LIN {X 0,Y 122.05,Z 340.248,A -85,B 0,C 180,E1 -25543.266,E2 -25543.266} C_VEL
LIN {X 0,Y 122.28,Z 340.237,A -85,B 0,C 180,E1 -25547.692,E2 -25547.692} C_VEL
LIN {X 0,Y 122.383,Z 340.24,A -85,B 0,C 180,E1 -25550.079,E2 -25550.079} C_VEL
LIN {X 0,Y 122.55,Z 340.186,A -85,B 0,C 180,E1 -25556.712,E2 -25556.712} C_VEL
LIN {X 0,Y 123.014,Z 340.16,A -85,B 0,C 180,E1 -25559.999,E2 -25559.999} C_VEL
LIN {X 0,Y 122.403,Z 340.204,A -85,B 0,C 180,E1 -25566.593,E2 -25566.593} C_VEL
LIN {X 0,Y 122.39,Z 340.237,A -85,B 0,C 180,E1 -25569.919,E2 -25569.919} C_VEL
LIN {X 0,Y 122.183,Z 340.246,A -85,B 0,C 180,E1 -25573.301,E2 -25573.301} C_VEL
LIN {X 0,Y 122.015,Z 340.287,A -85,B 0,C 180,E1 -25580.218,E2 -25580.218} C_VEL
LIN {X 0,Y 121.969,Z 340.291,A -85,B 0,C 180,E1 -25586.063,E2 -25586.063} C_VEL
LIN {X 0,Y 121.96,Z 340.291,A -85,B 0,C 180,E1 -25586.41,E2 -25586.41} C_VEL
LIN {X 0,Y 122.812,Z 342.955,A -85,B 0,C 180,E1 -25587.394,E2 -25587.394} C_VEL
LIN {X 0,Y 124.787,Z 345.128,A -85,B 0,C 180,E1 -25588.996,E2 -25588.996} C_VEL
LIN {X 0,Y 125.918,Z 346.004,A -85,B 0,C 180,E1 -25589.828,E2 -25589.828} C_VEL
LIN {X 0,Y 127.875,Z 349.273,A -85,B 0,C 180,E1 -25591.359,E2 -25591.359} C_VEL
LIN {X 0,Y 129.557,Z 351.048,A -85,B 0,C 180,E1 -25592.505,E2 -25592.505} C_VEL
LIN {X 0,Y 132.081,Z 354.649,A -85,B 0,C 180,E1 -25594.201,E2 -25594.201} C_VEL
LIN {X 0,Y 137.883,Z 363.38,A -85,B 0,C 180,E1 -25597.708,E2 -25597.708} C_VEL
LIN {X 0,Y 140.737,Z 368.366,A -85,B 0,C 180,E1 -25599.3,E2 -25599.3} C_VEL
LIN {X 0,Y 145.029,Z 378.064,A -85,B 0,C 180,E1 -25601.652,E2 -25601.652} C_VEL
LIN {X 0,Y 149.532,Z 390.716,A -85,B 0,C 180,E1 -25604.048,E2 -25604.048} C_VEL
LIN {X 0,Y 150.03,Z 393.35,A -85,B 0,C 180,E1 -25604.376,E2 -25604.376} C_VEL
LIN {X 0,Y 150.303,Z 399.971,A -85,B 0,C 180,E1 -25604.873,E2 -25604.873} C_VEL
LIN {X 0,Y 147.38,Z 443.847,A -85,B 0,C 180,E1 -25606.752,E2 -25606.752} C_VEL
LIN {X 0,Y 145.548,Z 457.609,A -85,B 0,C 180,E1 -25607.822,E2 -25607.822} C_VEL
LIN {X 0,Y 142.923,Z 470.589,A -85,B 0,C 180,E1 -25609.345,E2 -25609.345} C_VEL
LIN {X 0,Y 140.074,Z 481.613,A -85,B 0,C 180,E1 -25611.162,E2 -25611.162} C_VEL
LIN {X 0,Y 136.463,Z 493.143,A -85,B 0,C 180,E1 -25613.685,E2 -25613.685} C_VEL
LIN {X 0,Y 132.834,Z 503.54,A -85,B 0,C 180,E1 -25616.71,E2 -25616.71} C_VEL
LIN {X 0,Y 129.048,Z 513.69,A -85,B 0,C 180,E1 -25620.653,E2 -25620.653} C_VEL
LIN {X 0,Y 126.136,Z 521.23,A -85,B 0,C 180,E1 -25624.42,E2 -25624.42} C_VEL
LIN {X 0,Y 123.255,Z 528.616,A -85,B 0,C 180,E1 -25629.125,E2 -25629.125} C_VEL
LIN {X 0,Y 121.393,Z 533.602,A -85,B 0,C 180,E1 -25633.176,E2 -25633.176} C_VEL
LIN {X 0,Y 120.07,Z 538.442,A -85,B 0,C 180,E1 -25638.181,E2 -25638.181} C_VEL
LIN {X 0,Y 119.418,Z 542.133,A -85,B 0,C 180,E1 -25643.243,E2 -25643.243} C_VEL
LIN {X 0,Y 119.284,Z 544.029,A -85,B 0,C 180,E1 -25646.625,E2 -25646.625} C_VEL
LIN {X 0,Y 119.416,Z 545.463,A -85,B 0,C 180,E1 -25650.002,E2 -25650.002} C_VEL
LIN {X 0,Y 119.285,Z 546.45,A -85,B 0,C 180,E1 -25653.38,E2 -25653.38} C_VEL
LIN {X 0,Y 119.418,Z 547.051,A -85,B 0,C 180,E1 -25656.762,E2 -25656.762} C_VEL
LIN {X 0,Y 119.841,Z 547.27,A -85,B 0,C 180,E1 -25660.135,E2 -25660.135} C_VEL
LIN {X 0,Y 120.581,Z 547.087,A -85,B 0,C 180,E1 -25663.484,E2 -25663.484} C_VEL
LIN {X 0,Y 123.214,Z 545.523,A -85,B 0,C 180,E1 -25670.015,E2 -25670.015} C_VEL
LIN {X 0,Y 125.186,Z 544.168,A -85,B 0,C 180,E1 -25673.143,E2 -25673.143} C_VEL
LIN {X 0,Y 128.786,Z 541.327,A -85,B 0,C 180,E1 -25677.638,E2 -25677.638} C_VEL
LIN {X 0,Y 133.187,Z 537.486,A -85,B 0,C 180,E1 -25681.851,E2 -25681.851} C_VEL
LIN {X 0,Y 138.133,Z 532.546,A -85,B 0,C 180,E1 -25685.813,E2 -25685.813} C_VEL
LIN {X 0,Y 142.88,Z 527.3,A -85,B 0,C 180,E1 -25688.983,E2 -25688.983} C_VEL
LIN {X 0,Y 145.171,Z 524.1,A -85,B 0,C 180,E1 -25690.738,E2 -25690.738} C_VEL
LIN {X 0,Y 147.635,Z 518.574,A -85,B 0,C 180,E1 -25693.817,E2 -25693.817} C_VEL
LIN {X 0,Y 150.241,Z 512.543,A -85,B 0,C 180,E1 -25696.658,E2 -25696.658} C_VEL
LIN {X 0,Y 152.654,Z 508.469,A -85,B 0,C 180,E1 -25698.003,E2 -25698.003} C_VEL
LIN {X 0,Y 158.799,Z 498.626,A -85,B 0,C 180,E1 -25700.264,E2 -25700.264} C_VEL
LIN {X 0,Y 163.979,Z 488.786,A -85,B 0,C 180,E1 -25701.958,E2 -25701.958} C_VEL
LIN {X 0,Y 168.663,Z 478.109,A -85,B 0,C 180,E1 -25703.336,E2 -25703.336} C_VEL
LIN {X 0,Y 172.737,Z 466.399,A -85,B 0,C 180,E1 -25704.463,E2 -25704.463} C_VEL
LIN {X 0,Y 176.127,Z 453.278,A -85,B 0,C 180,E1 -25705.359,E2 -25705.359} C_VEL
LIN {X 0,Y 178.296,Z 439.911,A -85,B 0,C 180,E1 -25705.945,E2 -25705.945} C_VEL
LIN {X 0,Y 179.546,Z 425.717,A -85,B 0,C 180,E1 -25706.435,E2 -25706.435} C_VEL
LIN {X 0,Y 176.176,Z 416.595,A -85,B 0,C 180,E1 -25709.345,E2 -25709.345} C_VEL
LIN {X 0,Y 172.659,Z 408.352,A -85,B 0,C 180,E1 -25712.763,E2 -25712.763} C_VEL
LIN {X 0,Y 170.883,Z 404.467,A -85,B 0,C 180,E1 -25714.722,E2 -25714.722} C_VEL
LIN {X 0,Y 168.198,Z 398.886,A -85,B 0,C 180,E1 -25718.144,E2 -25718.144} C_VEL
LIN {X 0,Y 165.774,Z 394.965,A -85,B 0,C 180,E1 -25721.94,E2 -25721.94} C_VEL
LIN {X 0,Y 163.21,Z 390.77,A -85,B 0,C 180,E1 -25728.198,E2 -25728.198} C_VEL
LIN {X 0,Y 162.94,Z 389.949,A -85,B 0,C 180,E1 -25729.438,E2 -25729.438} C_VEL
LIN {X 0,Y 162.487,Z 389.493,A -85,B 0,C 180,E1 -25737.521,E2 -25737.521} C_VEL
LIN {X 0,Y 163.191,Z 389.938,A -85,B 0,C 180,E1 -25740.849,E2 -25740.849} C_VEL
LIN {X 0,Y 164.624,Z 393.257,A -85,B 0,C 180,E1 -25745.205,E2 -25745.205} C_VEL
LIN {X 0,Y 165.872,Z 394.947,A -85,B 0,C 180,E1 -25747.626,E2 -25747.626} C_VEL
LIN {X 0,Y 168.581,Z 399.566,A -85,B 0,C 180,E1 -25751.803,E2 -25751.803} C_VEL
LIN {X 0,Y 171.09,Z 403.702,A -85,B 0,C 180,E1 -25754.801,E2 -25754.801} C_VEL
LIN {X 0,Y 174.389,Z 409.476,A -85,B 0,C 180,E1 -25758.124,E2 -25758.124} C_VEL
LIN {X 0,Y 178.433,Z 417.155,A -85,B 0,C 180,E1 -25761.594,E2 -25761.594} C_VEL
LIN {X 0,Y 179.997,Z 420.592,A -85,B 0,C 180,E1 -25762.831,E2 -25762.831} C_VEL
LIN {X 0,Y 177.989,Z 440.073,A -85,B 0,C 180,E1 -25763.488,E2 -25763.488} C_VEL
LIN {X 0,Y 175.562,Z 452.452,A -85,B 0,C 180,E1 -25764.12,E2 -25764.12} C_VEL
LIN {X 0,Y 172.425,Z 464.153,A -85,B 0,C 180,E1 -25765.081,E2 -25765.081} C_VEL
LIN {X 0,Y 168.495,Z 475.082,A -85,B 0,C 180,E1 -25766.26,E2 -25766.26} C_VEL
LIN {X 0,Y 163.484,Z 486.45,A -85,B 0,C 180,E1 -25767.972,E2 -25767.972} C_VEL
LIN {X 0,Y 157.496,Z 497.496,A -85,B 0,C 180,E1 -25770.163,E2 -25770.163} C_VEL
LIN {X 0,Y 151.902,Z 506.082,A -85,B 0,C 180,E1 -25772.393,E2 -25772.393} C_VEL
LIN {X 0,Y 144.957,Z 515.194,A -85,B 0,C 180,E1 -25775.578,E2 -25775.578} C_VEL
LIN {X 0,Y 138.28,Z 522.741,A -85,B 0,C 180,E1 -25779.186,E2 -25779.186} C_VEL
LIN {X 0,Y 133.244,Z 527.718,A -85,B 0,C 180,E1 -25782.399,E2 -25782.399} C_VEL
LIN {X 0,Y 127.839,Z 532.518,A -85,B 0,C 180,E1 -25786.589,E2 -25786.589} C_VEL
LIN {X 0,Y 123.132,Z 536.152,A -85,B 0,C 180,E1 -25791.106,E2 -25791.106} C_VEL
LIN {X 0,Y 119.732,Z 538.422,A -85,B 0,C 180,E1 -25795.264,E2 -25795.264} C_VEL
LIN {X 0,Y 116.136,Z 540.307,A -85,B 0,C 180,E1 -25801.042,E2 -25801.042} C_VEL
LIN {X 0,Y 114.553,Z 540.859,A -85,B 0,C 180,E1 -25804.564,E2 -25804.564} C_VEL
LIN {X 0,Y 113.341,Z 540.951,A -85,B 0,C 180,E1 -25808.455,E2 -25808.455} C_VEL
LIN {X 0,Y 112.023,Z 539.967,A -85,B 0,C 180,E1 -25815.464,E2 -25815.464} C_VEL
LIN {X 0,Y 111.847,Z 538.873,A -85,B 0,C 180,E1 -25819.132,E2 -25819.132} C_VEL
LIN {X 0,Y 112,Z 537.319,A -85,B 0,C 180,E1 -25822.788,E2 -25822.788} C_VEL
LIN {X 0,Y 112.755,Z 534.417,A -85,B 0,C 180,E1 -25827.905,E2 -25827.905} C_VEL
LIN {X 0,Y 113.998,Z 530.051,A -85,B 0,C 180,E1 -25833.532,E2 -25833.532} C_VEL
LIN {X 0,Y 116.415,Z 523.712,A -85,B 0,C 180,E1 -25839.554,E2 -25839.554} C_VEL
LIN {X 0,Y 119.322,Z 516.818,A -85,B 0,C 180,E1 -25844.494,E2 -25844.494} C_VEL
LIN {X 0,Y 122.985,Z 508.179,A -85,B 0,C 180,E1 -25849.18,E2 -25849.18} C_VEL
LIN {X 0,Y 126.582,Z 499.324,A -85,B 0,C 180,E1 -25852.868,E2 -25852.868} C_VEL
LIN {X 0,Y 130.468,Z 489.549,A -85,B 0,C 180,E1 -25855.953,E2 -25855.953} C_VEL
LIN {X 0,Y 133.97,Z 478.877,A -85,B 0,C 180,E1 -25858.597,E2 -25858.597} C_VEL
LIN {X 0,Y 137.159,Z 466.941,A -85,B 0,C 180,E1 -25860.821,E2 -25860.821} C_VEL
LIN {X 0,Y 139.723,Z 454.541,A -85,B 0,C 180,E1 -25862.516,E2 -25862.516} C_VEL
LIN {X 0,Y 141.651,Z 441.546,A -85,B 0,C 180,E1 -25863.725,E2 -25863.725} C_VEL
LIN {X 0,Y 143.075,Z 424.971,A -85,B 0,C 180,E1 -25864.573,E2 -25864.573} C_VEL
LIN {X 0,Y 145.402,Z 390.427,A -85,B 0,C 180,E1 -25866.022,E2 -25866.022} C_VEL
LIN {X 0,Y 139.668,Z 378.184,A -85,B 0,C 180,E1 -25869.068,E2 -25869.068} C_VEL
LIN {X 0,Y 133.72,Z 367.749,A -85,B 0,C 180,E1 -25872.527,E2 -25872.527} C_VEL
LIN {X 0,Y 128.591,Z 360.025,A -85,B 0,C 180,E1 -25875.873,E2 -25875.873} C_VEL
LIN {X 0,Y 125.657,Z 355.95,A -85,B 0,C 180,E1 -25878,E2 -25878} C_VEL
LIN {X 0,Y 123.056,Z 352.211,A -85,B 0,C 180,E1 -25880.085,E2 -25880.085} C_VEL
LIN {X 0,Y 120.071,Z 348.913,A -85,B 0,C 180,E1 -25882.639,E2 -25882.639} C_VEL
LIN {X 0,Y 118.959,Z 346.749,A -85,B 0,C 180,E1 -25883.786,E2 -25883.786} C_VEL
LIN {X 0,Y 116.196,Z 344.608,A -85,B 0,C 180,E1 -25886.5,E2 -25886.5} C_VEL
LIN {X 0,Y 115.012,Z 342.226,A -85,B 0,C 180,E1 -25887.985,E2 -25887.985} C_VEL
LIN {X 0,Y 114.821,Z 341.175,A -85,B 0,C 180,E1 -25888.427,E2 -25888.427} C_VEL
LIN {X 0,Y 114.802,Z 341.148,A -85,B 0,C 180,E1 -25894.625,E2 -25894.625} C_VEL
LIN {X 0,Y 114.926,Z 341.167,A -85,B 0,C 180,E1 -25898.474,E2 -25898.474} C_VEL
LIN {X 0,Y 115.072,Z 341.116,A -85,B 0,C 180,E1 -25905.859,E2 -25905.859} C_VEL
LIN {X 0,Y 115.298,Z 341.121,A -85,B 0,C 180,E1 -25909.463,E2 -25909.463} C_VEL
LIN {X 0,Y 115.476,Z 341.065,A -85,B 0,C 180,E1 -25916.51,E2 -25916.51} C_VEL
LIN {X 0,Y 115.965,Z 341.038,A -85,B 0,C 180,E1 -25919.999,E2 -25919.999} C_VEL
LIN {X 0,Y 115.346,Z 341.084,A -85,B 0,C 180,E1 -25926.999,E2 -25926.999} C_VEL
LIN {X 0,Y 115.199,Z 341.123,A -85,B 0,C 180,E1 -25932.562,E2 -25932.562} C_VEL
LIN {X 0,Y 114.967,Z 341.174,A -85,B 0,C 180,E1 -25940.462,E2 -25940.462} C_VEL
LIN {X 0,Y 115.662,Z 343.507,A -85,B 0,C 180,E1 -25941.48,E2 -25941.48} C_VEL
LIN {X 0,Y 117.756,Z 345.988,A -85,B 0,C 180,E1 -25943.732,E2 -25943.732} C_VEL
LIN {X 0,Y 119.204,Z 346.968,A -85,B 0,C 180,E1 -25945.071,E2 -25945.071} C_VEL
LIN {X 0,Y 121.032,Z 350.151,A -85,B 0,C 180,E1 -25946.861,E2 -25946.861} C_VEL
LIN {X 0,Y 123.197,Z 352.402,A -85,B 0,C 180,E1 -25948.655,E2 -25948.655} C_VEL
LIN {X 0,Y 125.78,Z 356.037,A -85,B 0,C 180,E1 -25950.712,E2 -25950.712} C_VEL
LIN {X 0,Y 127.064,Z 357.855,A -85,B 0,C 180,E1 -25951.669,E2 -25951.669} C_VEL
LIN {X 0,Y 130.283,Z 362.559,A -85,B 0,C 180,E1 -25953.916,E2 -25953.916} C_VEL
LIN {X 0,Y 135.752,Z 371.145,A -85,B 0,C 180,E1 -25957.335,E2 -25957.335} C_VEL
LIN {X 0,Y 140.282,Z 381.573,A -85,B 0,C 180,E1 -25960.057,E2 -25960.057} C_VEL
LIN {X 0,Y 144.459,Z 393.679,A -85,B 0,C 180,E1 -25962.485,E2 -25962.485} C_VEL
LIN {X 0,Y 144.944,Z 399.765,A -85,B 0,C 180,E1 -25963.06,E2 -25963.06} C_VEL
LIN {X 0,Y 141.919,Z 443.257,A -85,B 0,C 180,E1 -25964.95,E2 -25964.95} C_VEL
LIN {X 0,Y 140.094,Z 456.812,A -85,B 0,C 180,E1 -25966.017,E2 -25966.017} C_VEL
LIN {X 0,Y 137.56,Z 468.886,A -85,B 0,C 180,E1 -25967.398,E2 -25967.398} C_VEL
LIN {X 0,Y 134.572,Z 480.296,A -85,B 0,C 180,E1 -25969.25,E2 -25969.25} C_VEL
LIN {X 0,Y 131.257,Z 490.735,A -85,B 0,C 180,E1 -25971.508,E2 -25971.508} C_VEL
LIN {X 0,Y 127.278,Z 501.504,A -85,B 0,C 180,E1 -25974.568,E2 -25974.568} C_VEL
LIN {X 0,Y 123.543,Z 511.223,A -85,B 0,C 180,E1 -25978.254,E2 -25978.254} C_VEL
LIN {X 0,Y 120.389,Z 519.177,A -85,B 0,C 180,E1 -25982.162,E2 -25982.162} C_VEL
LIN {X 0,Y 117.068,Z 526.893,A -85,B 0,C 180,E1 -25987.035,E2 -25987.035} C_VEL
LIN {X 0,Y 114.566,Z 533.083,A -85,B 0,C 180,E1 -25992.141,E2 -25992.141} C_VEL
LIN {X 0,Y 113.112,Z 537.994,A -85,B 0,C 180,E1 -25997.443,E2 -25997.443} C_VEL
LIN {X 0,Y 112.342,Z 541.747,A -85,B 0,C 180,E1 -26002.815,E2 -26002.815} C_VEL
LIN {X 0,Y 112.202,Z 543.674,A -85,B 0,C 180,E1 -26006.411,E2 -26006.411} C_VEL
LIN {X 0,Y 112.331,Z 545.165,A -85,B 0,C 180,E1 -26010.003,E2 -26010.003} C_VEL
LIN {X 0,Y 112.202,Z 546.182,A -85,B 0,C 180,E1 -26013.594,E2 -26013.594} C_VEL
LIN {X 0,Y 112.826,Z 547.057,A -85,B 0,C 180,E1 -26020.773,E2 -26020.773} C_VEL
LIN {X 0,Y 113.674,Z 546.921,A -85,B 0,C 180,E1 -26024.321,E2 -26024.321} C_VEL
LIN {X 0,Y 116.54,Z 545.422,A -85,B 0,C 180,E1 -26031.215,E2 -26031.215} C_VEL
LIN {X 0,Y 121.173,Z 542.372,A -85,B 0,C 180,E1 -26037.648,E2 -26037.648} C_VEL
LIN {X 0,Y 125.585,Z 538.931,A -85,B 0,C 180,E1 -26042.119,E2 -26042.119} C_VEL
LIN {X 0,Y 130.605,Z 534.436,A -85,B 0,C 180,E1 -26046.296,E2 -26046.296} C_VEL
LIN {X 0,Y 137.277,Z 527.664,A -85,B 0,C 180,E1 -26050.751,E2 -26050.751} C_VEL
LIN {X 0,Y 143.758,Z 520.325,A -85,B 0,C 180,E1 -26054.161,E2 -26054.161} C_VEL
LIN {X 0,Y 150.791,Z 511.238,A -85,B 0,C 180,E1 -26057.231,E2 -26057.231} C_VEL
LIN {X 0,Y 152.654,Z 508.469,A -85,B 0,C 180,E1 -26058.003,E2 -26058.003} C_VEL
LIN {X 0,Y 155.049,Z 504.252,A -85,B 0,C 180,E1 -26059.256,E2 -26059.256} C_VEL
LIN {X 0,Y 157.663,Z 497.141,A -85,B 0,C 180,E1 -26061.592,E2 -26061.592} C_VEL
LIN {X 0,Y 160.083,Z 489.616,A -85,B 0,C 180,E1 -26063.725,E2 -26063.725} C_VEL
LIN {X 0,Y 162.087,Z 484.679,A -85,B 0,C 180,E1 -26064.643,E2 -26064.643} C_VEL
LIN {X 0,Y 166.644,Z 473.877,A -85,B 0,C 180,E1 -26065.861,E2 -26065.861} C_VEL
LIN {X 0,Y 170.618,Z 461.527,A -85,B 0,C 180,E1 -26066.896,E2 -26066.896} C_VEL
LIN {X 0,Y 173.736,Z 448.119,A -85,B 0,C 180,E1 -26067.641,E2 -26067.641} C_VEL
LIN {X 0,Y 175.5,Z 434.788,A -85,B 0,C 180,E1 -26068.137,E2 -26068.137} C_VEL
LIN {X 0,Y 175.969,Z 428.609,A -85,B 0,C 180,E1 -26068.386,E2 -26068.386} C_VEL
LIN {X 0,Y 172.859,Z 420.02,A -85,B 0,C 180,E1 -26071.381,E2 -26071.381} C_VEL
LIN {X 0,Y 169.949,Z 412.743,A -85,B 0,C 180,E1 -26074.578,E2 -26074.578} C_VEL
LIN {X 0,Y 167.428,Z 407.201,A -85,B 0,C 180,E1 -26077.804,E2 -26077.804} C_VEL
LIN {X 0,Y 166.423,Z 405.138,A -85,B 0,C 180,E1 -26079.288,E2 -26079.288} C_VEL
LIN {X 0,Y 164.199,Z 401.326,A -85,B 0,C 180,E1 -26083.169,E2 -26083.169} C_VEL
LIN {X 0,Y 162.181,Z 397.615,A -85,B 0,C 180,E1 -26088.755,E2 -26088.755} C_VEL
LIN {X 0,Y 161.931,Z 396.919,A -85,B 0,C 180,E1 -26090.003,E2 -26090.003} C_VEL
LIN {X 0,Y 161.725,Z 396.564,A -85,B 0,C 180,E1 -26098.228,E2 -26098.228} C_VEL
LIN {X 0,Y 162.203,Z 396.945,A -85,B 0,C 180,E1 -26100.466,E2 -26100.466} C_VEL
LIN {X 0,Y 163.599,Z 400.242,A -85,B 0,C 180,E1 -26104.929,E2 -26104.929} C_VEL
LIN {X 0,Y 164.553,Z 401.63,A -85,B 0,C 180,E1 -26106.9,E2 -26106.9} C_VEL
LIN {X 0,Y 167.015,Z 406.088,A -85,B 0,C 180,E1 -26110.993,E2 -26110.993} C_VEL
LIN {X 0,Y 169.332,Z 410.145,A -85,B 0,C 180,E1 -26113.96,E2 -26113.96} C_VEL
LIN {X 0,Y 172.088,Z 415.151,A -85,B 0,C 180,E1 -26116.936,E2 -26116.936} C_VEL
LIN {X 0,Y 176.206,Z 423.49,A -85,B 0,C 180,E1 -26120.732,E2 -26120.732} C_VEL
LIN {X 0,Y 176.439,Z 424.028,A -85,B 0,C 180,E1 -26120.932,E2 -26120.932} C_VEL
LIN {X 0,Y 174.441,Z 441.483,A -85,B 0,C 180,E1 -26121.51,E2 -26121.51} C_VEL
LIN {X 0,Y 171.775,Z 454.185,A -85,B 0,C 180,E1 -26122.182,E2 -26122.182} C_VEL
LIN {X 0,Y 167.865,Z 467.297,A -85,B 0,C 180,E1 -26123.295,E2 -26123.295} C_VEL
LIN {X 0,Y 163.346,Z 478.817,A -85,B 0,C 180,E1 -26124.642,E2 -26124.642} C_VEL
LIN {X 0,Y 158.004,Z 489.815,A -85,B 0,C 180,E1 -26126.411,E2 -26126.411} C_VEL
LIN {X 0,Y 151.981,Z 499.889,A -85,B 0,C 180,E1 -26128.522,E2 -26128.522} C_VEL
LIN {X 0,Y 145.617,Z 508.928,A -85,B 0,C 180,E1 -26131.051,E2 -26131.051} C_VEL
LIN {X 0,Y 138.684,Z 517.33,A -85,B 0,C 180,E1 -26134.212,E2 -26134.212} C_VEL
LIN {X 0,Y 131.583,Z 524.614,A -85,B 0,C 180,E1 -26138.015,E2 -26138.015} C_VEL
LIN {X 0,Y 124.487,Z 530.95,A -85,B 0,C 180,E1 -26142.781,E2 -26142.781} C_VEL
LIN {X 0,Y 119.123,Z 535.036,A -85,B 0,C 180,E1 -26147.273,E2 -26147.273} C_VEL
LIN {X 0,Y 113.347,Z 538.705,A -85,B 0,C 180,E1 -26153.714,E2 -26153.714} C_VEL
LIN {X 0,Y 109.773,Z 540.425,A -85,B 0,C 180,E1 -26159.188,E2 -26159.188} C_VEL
LIN {X 0,Y 107.982,Z 541.012,A -85,B 0,C 180,E1 -26162.894,E2 -26162.894} C_VEL
LIN {X 0,Y 106.365,Z 541.14,A -85,B 0,C 180,E1 -26167.678,E2 -26167.678} C_VEL
LIN {X 0,Y 105.029,Z 540.255,A -85,B 0,C 180,E1 -26174.472,E2 -26174.472} C_VEL
LIN {X 0,Y 104.763,Z 539.201,A -85,B 0,C 180,E1 -26178.387,E2 -26178.387} C_VEL
LIN {X 0,Y 104.857,Z 537.712,A -85,B 0,C 180,E1 -26182.294,E2 -26182.294} C_VEL
LIN {X 0,Y 105.554,Z 535.228,A -85,B 0,C 180,E1 -26187.135,E2 -26187.135} C_VEL
LIN {X 0,Y 106.911,Z 530.591,A -85,B 0,C 180,E1 -26193.766,E2 -26193.766} C_VEL
LIN {X 0,Y 109.417,Z 524.337,A -85,B 0,C 180,E1 -26200.171,E2 -26200.171} C_VEL
LIN {X 0,Y 112.45,Z 517.538,A -85,B 0,C 180,E1 -26205.401,E2 -26205.401} C_VEL
LIN {X 0,Y 116.317,Z 509.064,A -85,B 0,C 180,E1 -26210.327,E2 -26210.327} C_VEL
LIN {X 0,Y 120.084,Z 500.345,A -85,B 0,C 180,E1 -26214.182,E2 -26214.182} C_VEL
LIN {X 0,Y 124.021,Z 490.76,A -85,B 0,C 180,E1 -26217.412,E2 -26217.412} C_VEL
LIN {X 0,Y 127.816,Z 480.285,A -85,B 0,C 180,E1 -26220.112,E2 -26220.112} C_VEL
LIN {X 0,Y 131.152,Z 468.802,A -85,B 0,C 180,E1 -26222.4,E2 -26222.4} C_VEL
LIN {X 0,Y 133.852,Z 456.913,A -85,B 0,C 180,E1 -26224.133,E2 -26224.133} C_VEL
LIN {X 0,Y 136.084,Z 443.206,A -85,B 0,C 180,E1 -26225.516,E2 -26225.516} C_VEL
LIN {X 0,Y 137.339,Z 430.812,A -85,B 0,C 180,E1 -26226.261,E2 -26226.261} C_VEL
LIN {X 0,Y 140.056,Z 392.687,A -85,B 0,C 180,E1 -26227.88,E2 -26227.88} C_VEL
LIN {X 0,Y 134.901,Z 381.566,A -85,B 0,C 180,E1 -26230.886,E2 -26230.886} C_VEL
LIN {X 0,Y 129.535,Z 372.061,A -85,B 0,C 180,E1 -26234.298,E2 -26234.298} C_VEL
LIN {X 0,Y 125.1,Z 365.244,A -85,B 0,C 180,E1 -26237.455,E2 -26237.455} C_VEL
LIN {X 0,Y 122.486,Z 361.454,A -85,B 0,C 180,E1 -26239.524,E2 -26239.524} C_VEL
LIN {X 0,Y 119.777,Z 357.638,A -85,B 0,C 180,E1 -26241.885,E2 -26241.885} C_VEL
LIN {X 0,Y 117.217,Z 354.408,A -85,B 0,C 180,E1 -26244.333,E2 -26244.333} C_VEL
LIN {X 0,Y 116.461,Z 353.066,A -85,B 0,C 180,E1 -26245.163,E2 -26245.163} C_VEL
LIN {X 0,Y 113.857,Z 350.628,A -85,B 0,C 180,E1 -26247.983,E2 -26247.983} C_VEL
LIN {X 0,Y 112.387,Z 347.844,A -85,B 0,C 180,E1 -26249.981,E2 -26249.981} C_VEL
LIN {X 0,Y 109.653,Z 346.082,A -85,B 0,C 180,E1 -26253.723,E2 -26253.723} C_VEL
LIN {X 0,Y 108.268,Z 343.712,A -85,B 0,C 180,E1 -26256.287,E2 -26256.287} C_VEL
LIN {X 0,Y 107.871,Z 342.033,A -85,B 0,C 180,E1 -26257.494,E2 -26257.494} C_VEL
LIN {X 0,Y 107.961,Z 341.997,A -85,B 0,C 180,E1 -26264.906,E2 -26264.906} C_VEL
LIN {X 0,Y 108.216,Z 341.998,A -85,B 0,C 180,E1 -26268.764,E2 -26268.764} C_VEL
LIN {X 0,Y 108.279,Z 341.973,A -85,B 0,C 180,E1 -26272.54,E2 -26272.54} C_VEL
LIN {X 0,Y 108.891,Z 341.919,A -85,B 0,C 180,E1 -26279.999,E2 -26279.999} C_VEL
LIN {X 0,Y 108.285,Z 341.965,A -85,B 0,C 180,E1 -26287.458,E2 -26287.458} C_VEL
LIN {X 0,Y 108.198,Z 342.025,A -85,B 0,C 180,E1 -26291.861,E2 -26291.861} C_VEL
LIN {X 0,Y 108.799,Z 344.324,A -85,B 0,C 180,E1 -26293.314,E2 -26293.314} C_VEL
LIN {X 0,Y 110.502,Z 346.638,A -85,B 0,C 180,E1 -26296.155,E2 -26296.155} C_VEL
LIN {X 0,Y 112.749,Z 348.094,A -85,B 0,C 180,E1 -26299.101,E2 -26299.101} C_VEL
LIN {X 0,Y 114.313,Z 351.012,A -85,B 0,C 180,E1 -26301.173,E2 -26301.173} C_VEL
LIN {X 0,Y 116.89,Z 353.611,A -85,B 0,C 180,E1 -26303.918,E2 -26303.918} C_VEL
LIN {X 0,Y 119.215,Z 357.045,A -85,B 0,C 180,E1 -26306.24,E2 -26306.24} C_VEL
LIN {X 0,Y 120.52,Z 358.544,A -85,B 0,C 180,E1 -26307.395,E2 -26307.395} C_VEL
LIN {X 0,Y 124.501,Z 364.347,A -85,B 0,C 180,E1 -26310.709,E2 -26310.709} C_VEL
LIN {X 0,Y 128.263,Z 370.003,A -85,B 0,C 180,E1 -26313.46,E2 -26313.46} C_VEL
LIN {X 0,Y 132.251,Z 376.864,A -85,B 0,C 180,E1 -26316.124,E2 -26316.124} C_VEL
LIN {X 0,Y 136.104,Z 386.284,A -85,B 0,C 180,E1 -26318.644,E2 -26318.644} C_VEL
LIN {X 0,Y 139.507,Z 396.653,A -85,B 0,C 180,E1 -26320.814,E2 -26320.814} C_VEL
LIN {X 0,Y 139.582,Z 402.148,A -85,B 0,C 180,E1 -26321.23,E2 -26321.23} C_VEL
LIN {X 0,Y 136.517,Z 443.449,A -85,B 0,C 180,E1 -26323.057,E2 -26323.057} C_VEL
LIN {X 0,Y 134.636,Z 456.775,A -85,B 0,C 180,E1 -26324.135,E2 -26324.135} C_VEL
LIN {X 0,Y 131.854,Z 469.366,A -85,B 0,C 180,E1 -26325.611,E2 -26325.611} C_VEL
LIN {X 0,Y 128.732,Z 480.582,A -85,B 0,C 180,E1 -26327.503,E2 -26327.503} C_VEL
LIN {X 0,Y 124.801,Z 492.239,A -85,B 0,C 180,E1 -26330.169,E2 -26330.169} C_VEL
LIN {X 0,Y 120.681,Z 502.718,A -85,B 0,C 180,E1 -26333.354,E2 -26333.354} C_VEL
LIN {X 0,Y 116.768,Z 512.141,A -85,B 0,C 180,E1 -26337.205,E2 -26337.205} C_VEL
LIN {X 0,Y 113.458,Z 519.883,A -85,B 0,C 180,E1 -26341.314,E2 -26341.314} C_VEL
LIN {X 0,Y 110.014,Z 527.43,A -85,B 0,C 180,E1 -26346.471,E2 -26346.471} C_VEL
LIN {X 0,Y 107.152,Z 534.387,A -85,B 0,C 180,E1 -26352.837,E2 -26352.837} C_VEL
LIN {X 0,Y 105.785,Z 538.963,A -85,B 0,C 180,E1 -26358.506,E2 -26358.506} C_VEL
LIN {X 0,Y 105.283,Z 541.362,A -85,B 0,C 180,E1 -26362.331,E2 -26362.331} C_VEL
LIN {X 0,Y 105.111,Z 543.32,A -85,B 0,C 180,E1 -26366.169,E2 -26366.169} C_VEL
LIN {X 0,Y 105.232,Z 544.854,A -85,B 0,C 180,E1 -26370.003,E2 -26370.003} C_VEL
LIN {X 0,Y 105.112,Z 545.913,A -85,B 0,C 180,E1 -26373.837,E2 -26373.837} C_VEL
LIN {X 0,Y 105.841,Z 546.843,A -85,B 0,C 180,E1 -26381.493,E2 -26381.493} C_VEL
LIN {X 0,Y 106.801,Z 546.74,A -85,B 0,C 180,E1 -26385.264,E2 -26385.264} C_VEL
LIN {X 0,Y 108.151,Z 546.236,A -85,B 0,C 180,E1 -26388.963,E2 -26388.963} C_VEL
LIN {X 0,Y 112.232,Z 544.023,A -85,B 0,C 180,E1 -26396.001,E2 -26396.001} C_VEL
LIN {X 0,Y 116.353,Z 541.302,A -85,B 0,C 180,E1 -26400.895,E2 -26400.895} C_VEL
LIN {X 0,Y 121.326,Z 537.588,A -85,B 0,C 180,E1 -26405.401,E2 -26405.401} C_VEL
LIN {X 0,Y 126.883,Z 532.786,A -85,B 0,C 180,E1 -26409.57,E2 -26409.57} C_VEL
LIN {X 0,Y 133.07,Z 526.753,A -85,B 0,C 180,E1 -26413.363,E2 -26413.363} C_VEL
LIN {X 0,Y 139.975,Z 519.263,A -85,B 0,C 180,E1 -26416.724,E2 -26416.724} C_VEL
LIN {X 0,Y 146.072,Z 511.636,A -85,B 0,C 180,E1 -26419.272,E2 -26419.272} C_VEL
LIN {X 0,Y 152.438,Z 502.393,A -85,B 0,C 180,E1 -26421.609,E2 -26421.609} C_VEL
LIN {X 0,Y 158.314,Z 492.142,A -85,B 0,C 180,E1 -26423.576,E2 -26423.576} C_VEL
LIN {X 0,Y 162.087,Z 484.679,A -85,B 0,C 180,E1 -26424.643,E2 -26424.643} C_VEL
LIN {X 0,Y 164.012,Z 479.628,A -85,B 0,C 180,E1 -26425.493,E2 -26425.493} C_VEL
LIN {X 0,Y 165.958,Z 471.251,A -85,B 0,C 180,E1 -26427.214,E2 -26427.214} C_VEL
LIN {X 0,Y 167.458,Z 462.549,A -85,B 0,C 180,E1 -26428.747,E2 -26428.747} C_VEL
LIN {X 0,Y 168.609,Z 456.994,A -85,B 0,C 180,E1 -26429.299,E2 -26429.299} C_VEL
LIN {X 0,Y 171.296,Z 443.775,A -85,B 0,C 180,E1 -26429.931,E2 -26429.931} C_VEL
LIN {X 0,Y 172.656,Z 431.847,A -85,B 0,C 180,E1 -26430.346,E2 -26430.346} C_VEL
LIN {X 0,Y 169.953,Z 423.974,A -85,B 0,C 180,E1 -26433.275,E2 -26433.275} C_VEL
LIN {X 0,Y 167.224,Z 416.916,A -85,B 0,C 180,E1 -26436.675,E2 -26436.675} C_VEL
LIN {X 0,Y 165.141,Z 411.961,A -85,B 0,C 180,E1 -26439.803,E2 -26439.803} C_VEL
LIN {X 0,Y 163.016,Z 408.16,A -85,B 0,C 180,E1 -26443.726,E2 -26443.726} C_VEL
LIN {X 0,Y 161.116,Z 404.213,A -85,B 0,C 180,E1 -26449.634,E2 -26449.634} C_VEL
LIN {X 0,Y 160.656,Z 403.702,A -85,B 0,C 180,E1 -26452.459,E2 -26452.459} C_VEL
LIN {X 0,Y 161.104,Z 403.741,A -85,B 0,C 180,E1 -26459.511,E2 -26459.511} C_VEL
LIN {X 0,Y 161.586,Z 405.348,A -85,B 0,C 180,E1 -26461.792,E2 -26461.792} C_VEL
LIN {X 0,Y 163.36,Z 408.499,A -85,B 0,C 180,E1 -26466.369,E2 -26466.369} C_VEL
LIN {X 0,Y 165.583,Z 412.811,A -85,B 0,C 180,E1 -26470.316,E2 -26470.316} C_VEL
LIN {X 0,Y 167.584,Z 416.516,A -85,B 0,C 180,E1 -26473.066,E2 -26473.066} C_VEL
LIN {X 0,Y 170.54,Z 422.339,A -85,B 0,C 180,E1 -26476.459,E2 -26476.459} C_VEL
LIN {X 0,Y 173.025,Z 427.558,A -85,B 0,C 180,E1 -26478.925,E2 -26478.925} C_VEL
LIN {X 0,Y 171.194,Z 442.453,A -85,B 0,C 180,E1 -26479.445,E2 -26479.445} C_VEL
LIN {X 0,Y 168.641,Z 454.043,A -85,B 0,C 180,E1 -26480.023,E2 -26480.023} C_VEL
LIN {X 0,Y 164.757,Z 466.842,A -85,B 0,C 180,E1 -26481.07,E2 -26481.07} C_VEL
LIN {X 0,Y 160.451,Z 477.689,A -85,B 0,C 180,E1 -26482.282,E2 -26482.282} C_VEL
LIN {X 0,Y 155.387,Z 488.05,A -85,B 0,C 180,E1 -26483.827,E2 -26483.827} C_VEL
LIN {X 0,Y 149.312,Z 498.308,A -85,B 0,C 180,E1 -26485.84,E2 -26485.84} C_VEL
LIN {X 0,Y 143.289,Z 506.782,A -85,B 0,C 180,E1 -26488.008,E2 -26488.008} C_VEL
LIN {X 0,Y 135.541,Z 516.03,A -85,B 0,C 180,E1 -26491.234,E2 -26491.234} C_VEL
LIN {X 0,Y 128.364,Z 523.341,A -85,B 0,C 180,E1 -26494.786,E2 -26494.786} C_VEL
LIN {X 0,Y 121.698,Z 529.175,A -85,B 0,C 180,E1 -26498.771,E2 -26498.771} C_VEL
LIN {X 0,Y 115.689,Z 533.722,A -85,B 0,C 180,E1 -26503.195,E2 -26503.195} C_VEL
LIN {X 0,Y 112.086,Z 536.104,A -85,B 0,C 180,E1 -26506.389,E2 -26506.389} C_VEL
LIN {X 0,Y 107.049,Z 538.995,A -85,B 0,C 180,E1 -26511.985,E2 -26511.985} C_VEL
LIN {X 0,Y 103.554,Z 540.544,A -85,B 0,C 180,E1 -26517.113,E2 -26517.113} C_VEL
LIN {X 0,Y 99.964,Z 541.389,A -85,B 0,C 180,E1 -26525.047,E2 -26525.047} C_VEL
LIN {X 0,Y 98.834,Z 541.172,A -85,B 0,C 180,E1 -26529.17,E2 -26529.17} C_VEL
LIN {X 0,Y 98.047,Z 540.544,A -85,B 0,C 180,E1 -26533.335,E2 -26533.335} C_VEL
LIN {X 0,Y 97.691,Z 539.523,A -85,B 0,C 180,E1 -26537.533,E2 -26537.533} C_VEL
LIN {X 0,Y 97.72,Z 538.098,A -85,B 0,C 180,E1 -26541.727,E2 -26541.727} C_VEL
LIN {X 0,Y 98.49,Z 535.37,A -85,B 0,C 180,E1 -26547.469,E2 -26547.469} C_VEL
LIN {X 0,Y 99.828,Z 531.114,A -85,B 0,C 180,E1 -26554.034,E2 -26554.034} C_VEL
LIN {X 0,Y 102.439,Z 524.96,A -85,B 0,C 180,E1 -26560.872,E2 -26560.872} C_VEL
LIN {X 0,Y 105.619,Z 518.255,A -85,B 0,C 180,E1 -26566.424,E2 -26566.424} C_VEL
LIN {X 0,Y 109.704,Z 509.929,A -85,B 0,C 180,E1 -26571.612,E2 -26571.612} C_VEL
LIN {X 0,Y 113.661,Z 501.359,A -85,B 0,C 180,E1 -26575.644,E2 -26575.644} C_VEL
LIN {X 0,Y 118.247,Z 490.765,A -85,B 0,C 180,E1 -26579.36,E2 -26579.36} C_VEL
LIN {X 0,Y 121.764,Z 481.668,A -85,B 0,C 180,E1 -26581.778,E2 -26581.778} C_VEL
LIN {X 0,Y 125.257,Z 470.492,A -85,B 0,C 180,E1 -26584.128,E2 -26584.128} C_VEL
LIN {X 0,Y 128.336,Z 457.972,A -85,B 0,C 180,E1 -26586.061,E2 -26586.061} C_VEL
LIN {X 0,Y 130.693,Z 444.534,A -85,B 0,C 180,E1 -26587.473,E2 -26587.473} C_VEL
LIN {X 0,Y 132.133,Z 431.622,A -85,B 0,C 180,E1 -26588.293,E2 -26588.293} C_VEL
LIN {X 0,Y 134.884,Z 395.035,A -85,B 0,C 180,E1 -26589.866,E2 -26589.866} C_VEL
LIN {X 0,Y 130.505,Z 385.503,A -85,B 0,C 180,E1 -26592.667,E2 -26592.667} C_VEL
LIN {X 0,Y 125.785,Z 376.91,A -85,B 0,C 180,E1 -26595.954,E2 -26595.954} C_VEL
LIN {X 0,Y 121.727,Z 370.416,A -85,B 0,C 180,E1 -26599.125,E2 -26599.125} C_VEL
LIN {X 0,Y 119.221,Z 366.73,A -85,B 0,C 180,E1 -26601.298,E2 -26601.298} C_VEL
LIN {X 0,Y 117.116,Z 363.62,A -85,B 0,C 180,E1 -26603.308,E2 -26603.308} C_VEL
LIN {X 0,Y 114.568,Z 360.07,A -85,B 0,C 180,E1 -26605.996,E2 -26605.996} C_VEL
LIN {X 0,Y 113.756,Z 359.087,A -85,B 0,C 180,E1 -26606.91,E2 -26606.91} C_VEL
LIN {X 0,Y 111.313,Z 356.145,A -85,B 0,C 180,E1 -26609.923,E2 -26609.923} C_VEL
LIN {X 0,Y 110.436,Z 354.477,A -85,B 0,C 180,E1 -26611.231,E2 -26611.231} C_VEL
LIN {X 0,Y 107.921,Z 352.543,A -85,B 0,C 180,E1 -26615.013,E2 -26615.013} C_VEL
LIN {X 0,Y 106.473,Z 349.767,A -85,B 0,C 180,E1 -26618.051,E2 -26618.051} C_VEL
LIN {X 0,Y 106.094,Z 348.921,A -85,B 0,C 180,E1 -26618.989,E2 -26618.989} C_VEL
LIN {X 0,Y 102.737,Z 346.454,A -85,B 0,C 180,E1 -26632.136,E2 -26632.136} C_VEL
LIN {X 0,Y 103.264,Z 346.379,A -85,B 0,C 180,E1 -26640.487,E2 -26640.487} C_VEL
LIN {X 0,Y 105.435,Z 348.496,A -85,B 0,C 180,E1 -26648.142,E2 -26648.142} C_VEL
LIN {X 0,Y 106.56,Z 349.064,A -85,B 0,C 180,E1 -26650.569,E2 -26650.569} C_VEL
LIN {X 0,Y 107.737,Z 351.889,A -85,B 0,C 180,E1 -26653.2,E2 -26653.2} C_VEL
LIN {X 0,Y 109.935,Z 354.097,A -85,B 0,C 180,E1 -26656.707,E2 -26656.707} C_VEL
LIN {X 0,Y 110.853,Z 354.917,A -85,B 0,C 180,E1 -26657.979,E2 -26657.979} C_VEL
LIN {X 0,Y 112.964,Z 358.201,A -85,B 0,C 180,E1 -26660.811,E2 -26660.811} C_VEL
LIN {X 0,Y 114.596,Z 359.988,A -85,B 0,C 180,E1 -26662.657,E2 -26662.657} C_VEL
LIN {X 0,Y 117.117,Z 363.548,A -85,B 0,C 180,E1 -26665.312,E2 -26665.312} C_VEL
LIN {X 0,Y 121.31,Z 369.722,A -85,B 0,C 180,E1 -26669.144,E2 -26669.144} C_VEL
LIN {X 0,Y 125.191,Z 375.902,A -85,B 0,C 180,E1 -26672.229,E2 -26672.229} C_VEL
LIN {X 0,Y 128.563,Z 382.032,A -85,B 0,C 180,E1 -26674.671,E2 -26674.671} C_VEL
LIN {X 0,Y 132.094,Z 391.319,A -85,B 0,C 180,E1 -26677.207,E2 -26677.207} C_VEL
LIN {X 0,Y 134.527,Z 399.408,A -85,B 0,C 180,E1 -26678.942,E2 -26678.942} C_VEL
LIN {X 0,Y 134.359,Z 404.188,A -85,B 0,C 180,E1 -26679.228,E2 -26679.228} C_VEL
LIN {X 0,Y 131.248,Z 443.904,A -85,B 0,C 180,E1 -26681.033,E2 -26681.033} C_VEL
LIN {X 0,Y 129.162,Z 457.475,A -85,B 0,C 180,E1 -26682.156,E2 -26682.156} C_VEL
LIN {X 0,Y 126.293,Z 469.791,A -85,B 0,C 180,E1 -26683.666,E2 -26683.666} C_VEL
LIN {X 0,Y 122.507,Z 482.461,A -85,B 0,C 180,E1 -26685.93,E2 -26685.93} C_VEL
LIN {X 0,Y 118.363,Z 493.729,A -85,B 0,C 180,E1 -26688.661,E2 -26688.661} C_VEL
LIN {X 0,Y 114.148,Z 503.855,A -85,B 0,C 180,E1 -26692.002,E2 -26692.002} C_VEL
LIN {X 0,Y 109.827,Z 513.526,A -85,B 0,C 180,E1 -26696.292,E2 -26696.292} C_VEL
LIN {X 0,Y 105.837,Z 521.939,A -85,B 0,C 180,E1 -26701.225,E2 -26701.225} C_VEL
LIN {X 0,Y 102.47,Z 529.055,A -85,B 0,C 180,E1 -26706.777,E2 -26706.777} C_VEL
LIN {X 0,Y 100.333,Z 533.88,A -85,B 0,C 180,E1 -26711.63,E2 -26711.63} C_VEL
LIN {X 0,Y 98.793,Z 538.531,A -85,B 0,C 180,E1 -26717.681,E2 -26717.681} C_VEL
LIN {X 0,Y 98.251,Z 540.977,A -85,B 0,C 180,E1 -26721.778,E2 -26721.778} C_VEL
LIN {X 0,Y 98.021,Z 542.965,A -85,B 0,C 180,E1 -26725.891,E2 -26725.891} C_VEL
LIN {X 0,Y 98.144,Z 544.531,A -85,B 0,C 180,E1 -26730.003,E2 -26730.003} C_VEL
LIN {X 0,Y 98.022,Z 545.644,A -85,B 0,C 180,E1 -26734.114,E2 -26734.114} C_VEL
LIN {X 0,Y 98.887,Z 546.63,A -85,B 0,C 180,E1 -26742.314,E2 -26742.314} C_VEL
LIN {X 0,Y 101.424,Z 546.099,A -85,B 0,C 180,E1 -26750.274,E2 -26750.274} C_VEL
LIN {X 0,Y 105.882,Z 543.955,A -85,B 0,C 180,E1 -26757.689,E2 -26757.689} C_VEL
LIN {X 0,Y 110.31,Z 541.296,A -85,B 0,C 180,E1 -26762.792,E2 -26762.792} C_VEL
LIN {X 0,Y 115.587,Z 537.647,A -85,B 0,C 180,E1 -26767.45,E2 -26767.45} C_VEL
LIN {X 0,Y 121.487,Z 532.915,A -85,B 0,C 180,E1 -26771.706,E2 -26771.706} C_VEL
LIN {X 0,Y 127.995,Z 526.958,A -85,B 0,C 180,E1 -26775.548,E2 -26775.548} C_VEL
LIN {X 0,Y 135.204,Z 519.554,A -85,B 0,C 180,E1 -26778.916,E2 -26778.916} C_VEL
LIN {X 0,Y 142.847,Z 510.361,A -85,B 0,C 180,E1 -26781.926,E2 -26781.926} C_VEL
LIN {X 0,Y 150.152,Z 499.777,A -85,B 0,C 180,E1 -26784.417,E2 -26784.417} C_VEL
LIN {X 0,Y 155.658,Z 490.298,A -85,B 0,C 180,E1 -26786.064,E2 -26786.064} C_VEL
LIN {X 0,Y 161.339,Z 478.501,A -85,B 0,C 180,E1 -26787.565,E2 -26787.565} C_VEL
LIN {X 0,Y 165.94,Z 466.164,A -85,B 0,C 180,E1 -26788.689,E2 -26788.689} C_VEL
LIN {X 0,Y 168.609,Z 456.994,A -85,B 0,C 180,E1 -26789.299,E2 -26789.299} C_VEL
LIN {X 0,Y 169.22,Z 453.238,A -85,B 0,C 180,E1 -26789.715,E2 -26789.715} C_VEL
LIN {X 0,Y 169.208,Z 447.406,A -85,B 0,C 180,E1 -26790.874,E2 -26790.874} C_VEL
LIN {X 0,Y 169.025,Z 441.512,A -85,B 0,C 180,E1 -26791.989,E2 -26791.989} C_VEL
LIN {X 0,Y 169.232,Z 437.662,A -85,B 0,C 180,E1 -26792.325,E2 -26792.325} C_VEL
LIN {X 0,Y 169.487,Z 434.94,A -85,B 0,C 180,E1 -26792.449,E2 -26792.449} C_VEL
LIN {X 0,Y 166.893,Z 427.074,A -85,B 0,C 180,E1 -26795.676,E2 -26795.676} C_VEL
LIN {X 0,Y 164.715,Z 421.114,A -85,B 0,C 180,E1 -26798.864,E2 -26798.864} C_VEL
LIN {X 0,Y 163.483,Z 418.253,A -85,B 0,C 180,E1 -26800.959,E2 -26800.959} C_VEL
LIN {X 0,Y 161.867,Z 415.009,A -85,B 0,C 180,E1 -26804.255,E2 -26804.255} C_VEL
LIN {X 0,Y 160.069,Z 410.982,A -85,B 0,C 180,E1 -26810.524,E2 -26810.524} C_VEL
LIN {X 0,Y 160.068,Z 410.711,A -85,B 0,C 180,E1 -26818.743,E2 -26818.743} C_VEL
LIN {X 0,Y 160.3,Z 411.211,A -85,B 0,C 180,E1 -26820,E2 -26820} C_VEL
LIN {X 0,Y 162.129,Z 415.272,A -85,B 0,C 180,E1 -26825.715,E2 -26825.715} C_VEL
LIN {X 0,Y 164.105,Z 419.336,A -85,B 0,C 180,E1 -26829.501,E2 -26829.501} C_VEL
LIN {X 0,Y 166.097,Z 423.32,A -85,B 0,C 180,E1 -26832.447,E2 -26832.447} C_VEL
LIN {X 0,Y 169.225,Z 429.895,A -85,B 0,C 180,E1 -26836.203,E2 -26836.203} C_VEL
LIN {X 0,Y 169.81,Z 431.277,A -85,B 0,C 180,E1 -26836.841,E2 -26836.841} C_VEL
LIN {X 0,Y 167.863,Z 444.737,A -85,B 0,C 180,E1 -26837.336,E2 -26837.336} C_VEL
LIN {X 0,Y 164.86,Z 457.215,A -85,B 0,C 180,E1 -26838.04,E2 -26838.04} C_VEL
LIN {X 0,Y 160.792,Z 469.442,A -85,B 0,C 180,E1 -26839.053,E2 -26839.053} C_VEL
LIN {X 0,Y 156.359,Z 479.791,A -85,B 0,C 180,E1 -26840.231,E2 -26840.231} C_VEL
LIN {X 0,Y 150.652,Z 490.627,A -85,B 0,C 180,E1 -26841.914,E2 -26841.914} C_VEL
LIN {X 0,Y 144.182,Z 500.644,A -85,B 0,C 180,E1 -26843.939,E2 -26843.939} C_VEL
LIN {X 0,Y 137.292,Z 509.621,A -85,B 0,C 180,E1 -26846.382,E2 -26846.382} C_VEL
LIN {X 0,Y 131.198,Z 516.41,A -85,B 0,C 180,E1 -26848.824,E2 -26848.824} C_VEL
LIN {X 0,Y 124.344,Z 523.074,A -85,B 0,C 180,E1 -26852.022,E2 -26852.022} C_VEL
LIN {X 0,Y 117.248,Z 529.018,A -85,B 0,C 180,E1 -26855.978,E2 -26855.978} C_VEL
LIN {X 0,Y 110.802,Z 533.658,A -85,B 0,C 180,E1 -26860.432,E2 -26860.432} C_VEL
LIN {X 0,Y 106.889,Z 536.083,A -85,B 0,C 180,E1 -26863.673,E2 -26863.673} C_VEL
LIN {X 0,Y 100.887,Z 539.276,A -85,B 0,C 180,E1 -26870.023,E2 -26870.023} C_VEL
LIN {X 0,Y 97.476,Z 540.664,A -85,B 0,C 180,E1 -26874.771,E2 -26874.771} C_VEL
LIN {X 0,Y 93.368,Z 541.577,A -85,B 0,C 180,E1 -26883.148,E2 -26883.148} C_VEL
LIN {X 0,Y 92.058,Z 541.424,A -85,B 0,C 180,E1 -26887.557,E2 -26887.557} C_VEL
LIN {X 0,Y 91.12,Z 540.831,A -85,B 0,C 180,E1 -26892.027,E2 -26892.027} C_VEL
LIN {X 0,Y 90.626,Z 539.843,A -85,B 0,C 180,E1 -26896.544,E2 -26896.544} C_VEL
LIN {X 0,Y 90.58,Z 538.458,A -85,B 0,C 180,E1 -26901.07,E2 -26901.07} C_VEL
LIN {X 0,Y 91.428,Z 535.491,A -85,B 0,C 180,E1 -26907.883,E2 -26907.883} C_VEL
LIN {X 0,Y 92.746,Z 531.607,A -85,B 0,C 180,E1 -26914.343,E2 -26914.343} C_VEL
LIN {X 0,Y 95.02,Z 526.548,A -85,B 0,C 180,E1 -26920.652,E2 -26920.652} C_VEL
LIN {X 0,Y 98.228,Z 520.188,A -85,B 0,C 180,E1 -26926.627,E2 -26926.627} C_VEL
LIN {X 0,Y 102.35,Z 512.23,A -85,B 0,C 180,E1 -26932.186,E2 -26932.186} C_VEL
LIN {X 0,Y 107.307,Z 502.335,A -85,B 0,C 180,E1 -26937.284,E2 -26937.284} C_VEL
LIN {X 0,Y 112.104,Z 491.928,A -85,B 0,C 180,E1 -26941.142,E2 -26941.142} C_VEL
LIN {X 0,Y 115.829,Z 483.028,A -85,B 0,C 180,E1 -26943.615,E2 -26943.615} C_VEL
LIN {X 0,Y 119.463,Z 472.135,A -85,B 0,C 180,E1 -26946.033,E2 -26946.033} C_VEL
LIN {X 0,Y 122.706,Z 460.111,A -85,B 0,C 180,E1 -26948,E2 -26948} C_VEL
LIN {X 0,Y 125.251,Z 447.322,A -85,B 0,C 180,E1 -26949.461,E2 -26949.461} C_VEL
LIN {X 0,Y 126.975,Z 433.48,A -85,B 0,C 180,E1 -26950.437,E2 -26950.437} C_VEL
LIN {X 0,Y 129.843,Z 397.431,A -85,B 0,C 180,E1 -26952.014,E2 -26952.014} C_VEL
LIN {X 0,Y 125.999,Z 388.915,A -85,B 0,C 180,E1 -26954.747,E2 -26954.747} C_VEL
LIN {X 0,Y 121.381,Z 380.259,A -85,B 0,C 180,E1 -26958.36,E2 -26958.36} C_VEL
LIN {X 0,Y 116.763,Z 372.905,A -85,B 0,C 180,E1 -26962.504,E2 -26962.504} C_VEL
LIN {X 0,Y 114.408,Z 369.432,A -85,B 0,C 180,E1 -26964.928,E2 -26964.928} C_VEL
LIN {X 0,Y 111.674,Z 365.483,A -85,B 0,C 180,E1 -26968.126,E2 -26968.126} C_VEL
LIN {X 0,Y 109.187,Z 362.21,A -85,B 0,C 180,E1 -26971.495,E2 -26971.495} C_VEL
LIN {X 0,Y 108.464,Z 361.041,A -85,B 0,C 180,E1 -26972.635,E2 -26972.635} C_VEL
LIN {X 0,Y 106.064,Z 358.723,A -85,B 0,C 180,E1 -26976.713,E2 -26976.713} C_VEL
LIN {X 0,Y 104.763,Z 355.845,A -85,B 0,C 180,E1 -26979.906,E2 -26979.906} C_VEL
LIN {X 0,Y 101.867,Z 353.525,A -85,B 0,C 180,E1 -26992.068,E2 -26992.068} C_VEL
LIN {X 0,Y 102.303,Z 353.382,A -85,B 0,C 180,E1 -26999.999,E2 -26999.999} C_VEL
LIN {X 0,Y 104.001,Z 355.272,A -85,B 0,C 180,E1 -27006.791,E2 -27006.791} C_VEL
LIN {X 0,Y 105.068,Z 355.925,A -85,B 0,C 180,E1 -27009.383,E2 -27009.383} C_VEL
LIN {X 0,Y 106.702,Z 359.259,A -85,B 0,C 180,E1 -27013.085,E2 -27013.085} C_VEL
LIN {X 0,Y 108.977,Z 361.503,A -85,B 0,C 180,E1 -27016.749,E2 -27016.749} C_VEL
LIN {X 0,Y 111.334,Z 364.98,A -85,B 0,C 180,E1 -27020.074,E2 -27020.074} C_VEL
LIN {X 0,Y 112.485,Z 366.491,A -85,B 0,C 180,E1 -27021.489,E2 -27021.489} C_VEL
LIN {X 0,Y 115.617,Z 371.111,A -85,B 0,C 180,E1 -27024.966,E2 -27024.966} C_VEL
LIN {X 0,Y 119.72,Z 377.476,A -85,B 0,C 180,E1 -27028.846,E2 -27028.846} C_VEL
LIN {X 0,Y 124.442,Z 385.939,A -85,B 0,C 180,E1 -27032.717,E2 -27032.717} C_VEL
LIN {X 0,Y 127.634,Z 394.636,A -85,B 0,C 180,E1 -27035.26,E2 -27035.26} C_VEL
LIN {X 0,Y 129.643,Z 401.364,A -85,B 0,C 180,E1 -27036.837,E2 -27036.837} C_VEL
LIN {X 0,Y 126.243,Z 443.625,A -85,B 0,C 180,E1 -27038.8,E2 -27038.8} C_VEL
LIN {X 0,Y 124.023,Z 457.356,A -85,B 0,C 180,E1 -27039.939,E2 -27039.939} C_VEL
LIN {X 0,Y 121.182,Z 469.133,A -85,B 0,C 180,E1 -27041.387,E2 -27041.387} C_VEL
LIN {X 0,Y 117.465,Z 481.105,A -85,B 0,C 180,E1 -27043.498,E2 -27043.498} C_VEL
LIN {X 0,Y 113.139,Z 492.597,A -85,B 0,C 180,E1 -27046.29,E2 -27046.29} C_VEL
LIN {X 0,Y 108.577,Z 502.934,A -85,B 0,C 180,E1 -27049.667,E2 -27049.667} C_VEL
LIN {X 0,Y 104.27,Z 512.049,A -85,B 0,C 180,E1 -27053.736,E2 -27053.736} C_VEL
LIN {X 0,Y 100.412,Z 519.887,A -85,B 0,C 180,E1 -27058.34,E2 -27058.34} C_VEL
LIN {X 0,Y 96.502,Z 527.365,A -85,B 0,C 180,E1 -27064.093,E2 -27064.093} C_VEL
LIN {X 0,Y 93.576,Z 533.354,A -85,B 0,C 180,E1 -27070.25,E2 -27070.25} C_VEL
LIN {X 0,Y 91.835,Z 538.078,A -85,B 0,C 180,E1 -27076.731,E2 -27076.731} C_VEL
LIN {X 0,Y 91.014,Z 541.658,A -85,B 0,C 180,E1 -27083.352,E2 -27083.352} C_VEL
LIN {X 0,Y 91.048,Z 544.203,A -85,B 0,C 180,E1 -27090.003,E2 -27090.003} C_VEL
LIN {X 0,Y 90.931,Z 545.362,A -85,B 0,C 180,E1 -27094.436,E2 -27094.436} C_VEL
LIN {X 0,Y 91.225,Z 546.085,A -85,B 0,C 180,E1 -27098.867,E2 -27098.867} C_VEL
LIN {X 0,Y 93.105,Z 546.37,A -85,B 0,C 180,E1 -27107.577,E2 -27107.577} C_VEL
LIN {X 0,Y 94.76,Z 545.948,A -85,B 0,C 180,E1 -27111.77,E2 -27111.77} C_VEL
LIN {X 0,Y 96.939,Z 545.125,A -85,B 0,C 180,E1 -27115.788,E2 -27115.788} C_VEL
LIN {X 0,Y 102.699,Z 542.255,A -85,B 0,C 180,E1 -27123.196,E2 -27123.196} C_VEL
LIN {X 0,Y 108.104,Z 539.002,A -85,B 0,C 180,E1 -27128.145,E2 -27128.145} C_VEL
LIN {X 0,Y 114.107,Z 534.71,A -85,B 0,C 180,E1 -27132.652,E2 -27132.652} C_VEL
LIN {X 0,Y 121.945,Z 528.254,A -85,B 0,C 180,E1 -27137.294,E2 -27137.294} C_VEL
LIN {X 0,Y 129.348,Z 521.196,A -85,B 0,C 180,E1 -27140.741,E2 -27140.741} C_VEL
LIN {X 0,Y 137.254,Z 512.413,A -85,B 0,C 180,E1 -27143.755,E2 -27143.755} C_VEL
LIN {X 0,Y 144.751,Z 502.462,A -85,B 0,C 180,E1 -27146.252,E2 -27146.252} C_VEL
LIN {X 0,Y 151.088,Z 492.318,A -85,B 0,C 180,E1 -27148.097,E2 -27148.097} C_VEL
LIN {X 0,Y 156.934,Z 481.072,A -85,B 0,C 180,E1 -27149.553,E2 -27149.553} C_VEL
LIN {X 0,Y 162.095,Z 468.472,A -85,B 0,C 180,E1 -27150.745,E2 -27150.745} C_VEL
LIN {X 0,Y 165.986,Z 455.44,A -85,B 0,C 180,E1 -27151.601,E2 -27151.601} C_VEL
LIN {X 0,Y 168.521,Z 443,A -85,B 0,C 180,E1 -27152.143,E2 -27152.143} C_VEL
LIN {X 0,Y 169.232,Z 437.662,A -85,B 0,C 180,E1 -27152.325,E2 -27152.325} C_VEL
LIN {X 0,Y 169.282,Z 435.126,A -85,B 0,C 180,E1 -27152.608,E2 -27152.608} C_VEL
LIN {X 0,Y 168.767,Z 432.347,A -85,B 0,C 180,E1 -27153.388,E2 -27153.388} C_VEL
LIN {X 0,Y 167.599,Z 429.837,A -85,B 0,C 180,E1 -27154.743,E2 -27154.743} C_VEL
LIN {X 0,Y 166.491,Z 428.559,A -85,B 0,C 180,E1 -27155.963,E2 -27155.963} C_VEL
LIN {X 0,Y 162.344,Z 425.283,A -85,B 0,C 180,E1 -27161.314,E2 -27161.314} C_VEL
LIN {X 0,Y 161.931,Z 424.554,A -85,B 0,C 180,E1 -27162.076,E2 -27162.076} C_VEL
LIN {X 0,Y 160.616,Z 421.726,A -85,B 0,C 180,E1 -27165.06,E2 -27165.06} C_VEL
LIN {X 0,Y 159.172,Z 418.029,A -85,B 0,C 180,E1 -27170.63,E2 -27170.63} C_VEL
LIN {X 0,Y 159.193,Z 417.758,A -85,B 0,C 180,E1 -27178.736,E2 -27178.736} C_VEL
LIN {X 0,Y 160.906,Z 421.987,A -85,B 0,C 180,E1 -27185.012,E2 -27185.012} C_VEL
LIN {X 0,Y 162.753,Z 426.13,A -85,B 0,C 180,E1 -27188.85,E2 -27188.85} C_VEL
LIN {X 0,Y 164.499,Z 429.853,A -85,B 0,C 180,E1 -27191.631,E2 -27191.631} C_VEL
LIN {X 0,Y 166.788,Z 435.143,A -85,B 0,C 180,E1 -27194.723,E2 -27194.723} C_VEL
LIN {X 0,Y 164.515,Z 448.217,A -85,B 0,C 180,E1 -27195.22,E2 -27195.22} C_VEL
LIN {X 0,Y 161.269,Z 460.271,A -85,B 0,C 180,E1 -27195.945,E2 -27195.945} C_VEL
LIN {X 0,Y 157.026,Z 471.827,A -85,B 0,C 180,E1 -27196.923,E2 -27196.923} C_VEL
LIN {X 0,Y 151.729,Z 483.193,A -85,B 0,C 180,E1 -27198.273,E2 -27198.273} C_VEL
LIN {X 0,Y 145.659,Z 493.793,A -85,B 0,C 180,E1 -27199.999,E2 -27199.999} C_VEL
LIN {X 0,Y 138.485,Z 503.903,A -85,B 0,C 180,E1 -27202.15,E2 -27202.15} C_VEL
LIN {X 0,Y 131.416,Z 512.302,A -85,B 0,C 180,E1 -27204.608,E2 -27204.608} C_VEL
LIN {X 0,Y 123.262,Z 520.487,A -85,B 0,C 180,E1 -27207.897,E2 -27207.897} C_VEL
LIN {X 0,Y 115.537,Z 527.001,A -85,B 0,C 180,E1 -27211.61,E2 -27211.61} C_VEL
LIN {X 0,Y 109.1,Z 531.688,A -85,B 0,C 180,E1 -27215.435,E2 -27215.435} C_VEL
LIN {X 0,Y 101.955,Z 536.062,A -85,B 0,C 180,E1 -27220.685,E2 -27220.685} C_VEL
LIN {X 0,Y 94.848,Z 539.56,A -85,B 0,C 180,E1 -27227.816,E2 -27227.816} C_VEL
LIN {X 0,Y 91.591,Z 540.784,A -85,B 0,C 180,E1 -27232.128,E2 -27232.128} C_VEL
LIN {X 0,Y 86.895,Z 541.764,A -85,B 0,C 180,E1 -27240.966,E2 -27240.966} C_VEL
LIN {X 0,Y 85.37,Z 541.659,A -85,B 0,C 180,E1 -27245.69,E2 -27245.69} C_VEL
LIN {X 0,Y 84.251,Z 541.117,A -85,B 0,C 180,E1 -27250.505,E2 -27250.505} C_VEL
LIN {X 0,Y 83.592,Z 540.163,A -85,B 0,C 180,E1 -27255.387,E2 -27255.387} C_VEL
LIN {X 0,Y 83.47,Z 538.81,A -85,B 0,C 180,E1 -27260.302,E2 -27260.302} C_VEL
LIN {X 0,Y 84.376,Z 535.648,A -85,B 0,C 180,E1 -27268.287,E2 -27268.287} C_VEL
LIN {X 0,Y 85.665,Z 532.098,A -85,B 0,C 180,E1 -27274.702,E2 -27274.702} C_VEL
LIN {X 0,Y 88.052,Z 527.117,A -85,B 0,C 180,E1 -27281.507,E2 -27281.507} C_VEL
LIN {X 0,Y 91.465,Z 520.862,A -85,B 0,C 180,E1 -27287.896,E2 -27287.896} C_VEL
LIN {X 0,Y 95.819,Z 513.037,A -85,B 0,C 180,E1 -27293.788,E2 -27293.788} C_VEL
LIN {X 0,Y 101.062,Z 503.265,A -85,B 0,C 180,E1 -27299.126,E2 -27299.126} C_VEL
LIN {X 0,Y 106.097,Z 493.09,A -85,B 0,C 180,E1 -27303.123,E2 -27303.123} C_VEL
LIN {X 0,Y 110.556,Z 482.966,A -85,B 0,C 180,E1 -27306.013,E2 -27306.013} C_VEL
LIN {X 0,Y 114.388,Z 472.014,A -85,B 0,C 180,E1 -27308.464,E2 -27308.464} C_VEL
LIN {X 0,Y 117.801,Z 459.903,A -85,B 0,C 180,E1 -27310.447,E2 -27310.447} C_VEL
LIN {X 0,Y 120.422,Z 447.223,A -85,B 0,C 180,E1 -27311.883,E2 -27311.883} C_VEL
LIN {X 0,Y 122.121,Z 434.266,A -85,B 0,C 180,E1 -27312.812,E2 -27312.812} C_VEL
LIN {X 0,Y 125.04,Z 399.958,A -85,B 0,C 180,E1 -27314.298,E2 -27314.298} C_VEL
LIN {X 0,Y 121.347,Z 391.753,A -85,B 0,C 180,E1 -27317.244,E2 -27317.244} C_VEL
LIN {X 0,Y 117.301,Z 384.11,A -85,B 0,C 180,E1 -27320.817,E2 -27320.817} C_VEL
LIN {X 0,Y 113.676,Z 378.106,A -85,B 0,C 180,E1 -27324.481,E2 -27324.481} C_VEL
LIN {X 0,Y 111.891,Z 375.33,A -85,B 0,C 180,E1 -27326.52,E2 -27326.52} C_VEL
LIN {X 0,Y 109.558,Z 371.752,A -85,B 0,C 180,E1 -27329.506,E2 -27329.506} C_VEL
LIN {X 0,Y 107.099,Z 368.179,A -85,B 0,C 180,E1 -27333.205,E2 -27333.205} C_VEL
LIN {X 0,Y 104.224,Z 364.711,A -85,B 0,C 180,E1 -27338.674,E2 -27338.674} C_VEL
LIN {X 0,Y 103.473,Z 362.829,A -85,B 0,C 180,E1 -27340.795,E2 -27340.795} C_VEL
LIN {X 0,Y 100.997,Z 360.596,A -85,B 0,C 180,E1 -27351.999,E2 -27351.999} C_VEL
LIN {X 0,Y 101.275,Z 360.384,A -85,B 0,C 180,E1 -27359.005,E2 -27359.005} C_VEL
LIN {X 0,Y 103.696,Z 362.828,A -85,B 0,C 180,E1 -27368.341,E2 -27368.341} C_VEL
LIN {X 0,Y 105.497,Z 366.321,A -85,B 0,C 180,E1 -27372.626,E2 -27372.626} C_VEL
LIN {X 0,Y 107.205,Z 368.117,A -85,B 0,C 180,E1 -27375.561,E2 -27375.561} C_VEL
LIN {X 0,Y 110.326,Z 372.807,A -85,B 0,C 180,E1 -27380.144,E2 -27380.144} C_VEL
LIN {X 0,Y 113.284,Z 377.393,A -85,B 0,C 180,E1 -27383.707,E2 -27383.707} C_VEL
LIN {X 0,Y 116.695,Z 382.912,A -85,B 0,C 180,E1 -27387.215,E2 -27387.215} C_VEL
LIN {X 0,Y 120.932,Z 391.053,A -85,B 0,C 180,E1 -27391.049,E2 -27391.049} C_VEL
LIN {X 0,Y 123.908,Z 399.978,A -85,B 0,C 180,E1 -27393.696,E2 -27393.696} C_VEL
LIN {X 0,Y 124.835,Z 403.215,A -85,B 0,C 180,E1 -27394.506,E2 -27394.506} C_VEL
LIN {X 0,Y 121.441,Z 443.313,A -85,B 0,C 180,E1 -27396.381,E2 -27396.381} C_VEL
LIN {X 0,Y 119.169,Z 456.963,A -85,B 0,C 180,E1 -27397.522,E2 -27397.522} C_VEL
LIN {X 0,Y 115.971,Z 469.505,A -85,B 0,C 180,E1 -27399.068,E2 -27399.068} C_VEL
LIN {X 0,Y 112.071,Z 481.347,A -85,B 0,C 180,E1 -27401.195,E2 -27401.195} C_VEL
LIN {X 0,Y 107.515,Z 492.757,A -85,B 0,C 180,E1 -27404.029,E2 -27404.029} C_VEL
LIN {X 0,Y 102.725,Z 503.016,A -85,B 0,C 180,E1 -27407.503,E2 -27407.503} C_VEL
LIN {X 0,Y 98.331,Z 511.721,A -85,B 0,C 180,E1 -27411.525,E2 -27411.525} C_VEL
LIN {X 0,Y 94.403,Z 519.193,A -85,B 0,C 180,E1 -27416.062,E2 -27416.062} C_VEL
LIN {X 0,Y 90.137,Z 526.759,A -85,B 0,C 180,E1 -27422.111,E2 -27422.111} C_VEL
LIN {X 0,Y 86.868,Z 532.824,A -85,B 0,C 180,E1 -27428.654,E2 -27428.654} C_VEL
LIN {X 0,Y 84.917,Z 537.62,A -85,B 0,C 180,E1 -27435.627,E2 -27435.627} C_VEL
LIN {X 0,Y 83.958,Z 541.266,A -85,B 0,C 180,E1 -27442.79,E2 -27442.79} C_VEL
LIN {X 0,Y 83.945,Z 543.872,A -85,B 0,C 180,E1 -27450.003,E2 -27450.003} C_VEL
LIN {X 0,Y 83.864,Z 545.065,A -85,B 0,C 180,E1 -27454.811,E2 -27454.811} C_VEL
LIN {X 0,Y 84.199,Z 545.842,A -85,B 0,C 180,E1 -27459.613,E2 -27459.613} C_VEL
LIN {X 0,Y 86.336,Z 546.185,A -85,B 0,C 180,E1 -27469.006,E2 -27469.006} C_VEL
LIN {X 0,Y 90.591,Z 545.02,A -85,B 0,C 180,E1 -27477.744,E2 -27477.744} C_VEL
LIN {X 0,Y 96.819,Z 542.218,A -85,B 0,C 180,E1 -27485.504,E2 -27485.504} C_VEL
LIN {X 0,Y 102.601,Z 539.028,A -85,B 0,C 180,E1 -27490.6,E2 -27490.6} C_VEL
LIN {X 0,Y 108.975,Z 534.803,A -85,B 0,C 180,E1 -27495.19,E2 -27495.19} C_VEL
LIN {X 0,Y 117.238,Z 528.42,A -85,B 0,C 180,E1 -27499.849,E2 -27499.849} C_VEL
LIN {X 0,Y 124.984,Z 521.479,A -85,B 0,C 180,E1 -27503.257,E2 -27503.257} C_VEL
LIN {X 0,Y 133.192,Z 512.802,A -85,B 0,C 180,E1 -27506.211,E2 -27506.211} C_VEL
LIN {X 0,Y 140.267,Z 503.938,A -85,B 0,C 180,E1 -27508.408,E2 -27508.408} C_VEL
LIN {X 0,Y 147.476,Z 493.044,A -85,B 0,C 180,E1 -27510.428,E2 -27510.428} C_VEL
LIN {X 0,Y 153.48,Z 482.011,A -85,B 0,C 180,E1 -27511.824,E2 -27511.824} C_VEL
LIN {X 0,Y 158.81,Z 469.616,A -85,B 0,C 180,E1 -27512.974,E2 -27512.974} C_VEL
LIN {X 0,Y 162.819,Z 457.253,A -85,B 0,C 180,E1 -27513.772,E2 -27513.772} C_VEL
LIN {X 0,Y 165.607,Z 444.584,A -85,B 0,C 180,E1 -27514.344,E2 -27514.344} C_VEL
LIN {X 0,Y 166.49,Z 438.161,A -85,B 0,C 180,E1 -27514.617,E2 -27514.617} C_VEL
LIN {X 0,Y 164.02,Z 430.081,A -85,B 0,C 180,E1 -27518.311,E2 -27518.311} C_VEL
LIN {X 0,Y 162.31,Z 425.215,A -85,B 0,C 180,E1 -27521.372,E2 -27521.372} C_VEL
LIN {X 0,Y 161.931,Z 424.554,A -85,B 0,C 180,E1 -27522.076,E2 -27522.076} C_VEL
LIN {X 0,Y 160.924,Z 423.232,A -85,B 0,C 180,E1 -27524.08,E2 -27524.08} C_VEL
LIN {X 0,Y 159.946,Z 423.056,A -85,B 0,C 180,E1 -27526.169,E2 -27526.169} C_VEL
LIN {X 0,Y 158.124,Z 424.702,A -85,B 0,C 180,E1 -27531.914,E2 -27531.914} C_VEL
LIN {X 0,Y 157.954,Z 424.838,A -85,B 0,C 180,E1 -27533.379,E2 -27533.379} C_VEL
LIN {X 0,Y 158.316,Z 424.816,A -85,B 0,C 180,E1 -27538.729,E2 -27538.729} C_VEL
LIN {X 0,Y 159.745,Z 428.857,A -85,B 0,C 180,E1 -27544.416,E2 -27544.416} C_VEL
LIN {X 0,Y 161.401,Z 432.815,A -85,B 0,C 180,E1 -27548.136,E2 -27548.136} C_VEL
LIN {X 0,Y 163.099,Z 436.913,A -85,B 0,C 180,E1 -27551.181,E2 -27551.181} C_VEL
LIN {X 0,Y 163.887,Z 439.263,A -85,B 0,C 180,E1 -27552.539,E2 -27552.539} C_VEL
LIN {X 0,Y 160.939,Z 453.01,A -85,B 0,C 180,E1 -27553.093,E2 -27553.093} C_VEL
LIN {X 0,Y 157.054,Z 465.49,A -85,B 0,C 180,E1 -27553.948,E2 -27553.948} C_VEL
LIN {X 0,Y 151.93,Z 477.53,A -85,B 0,C 180,E1 -27555.058,E2 -27555.058} C_VEL
LIN {X 0,Y 145.691,Z 489.189,A -85,B 0,C 180,E1 -27556.604,E2 -27556.604} C_VEL
LIN {X 0,Y 138.911,Z 499.406,A -85,B 0,C 180,E1 -27558.44,E2 -27558.44} C_VEL
LIN {X 0,Y 131.453,Z 508.654,A -85,B 0,C 180,E1 -27560.667,E2 -27560.667} C_VEL
LIN {X 0,Y 122.798,Z 517.63,A -85,B 0,C 180,E1 -27563.688,E2 -27563.688} C_VEL
LIN {X 0,Y 114.544,Z 524.752,A -85,B 0,C 180,E1 -27567.164,E2 -27567.164} C_VEL
LIN {X 0,Y 106.766,Z 530.402,A -85,B 0,C 180,E1 -27571.154,E2 -27571.154} C_VEL
LIN {X 0,Y 99.583,Z 534.804,A -85,B 0,C 180,E1 -27575.743,E2 -27575.743} C_VEL
LIN {X 0,Y 93.132,Z 538.087,A -85,B 0,C 180,E1 -27581.003,E2 -27581.003} C_VEL
LIN {X 0,Y 88.935,Z 539.854,A -85,B 0,C 180,E1 -27585.336,E2 -27585.336} C_VEL
LIN {X 0,Y 85.925,Z 540.895,A -85,B 0,C 180,E1 -27589.127,E2 -27589.127} C_VEL
LIN {X 0,Y 82.983,Z 541.626,A -85,B 0,C 180,E1 -27593.637,E2 -27593.637} C_VEL
LIN {X 0,Y 78.761,Z 541.881,A -85,B 0,C 180,E1 -27603.499,E2 -27603.499} C_VEL
LIN {X 0,Y 77.423,Z 541.404,A -85,B 0,C 180,E1 -27608.706,E2 -27608.706} C_VEL
LIN {X 0,Y 76.597,Z 540.484,A -85,B 0,C 180,E1 -27614.019,E2 -27614.019} C_VEL
LIN {X 0,Y 76.357,Z 539.164,A -85,B 0,C 180,E1 -27619.389,E2 -27619.389} C_VEL
LIN {X 0,Y 77.326,Z 535.78,A -85,B 0,C 180,E1 -27628.826,E2 -27628.826} C_VEL
LIN {X 0,Y 79.245,Z 531.1,A -85,B 0,C 180,E1 -27637.641,E2 -27637.641} C_VEL
LIN {X 0,Y 82.767,Z 524.775,A -85,B 0,C 180,E1 -27646.016,E2 -27646.016} C_VEL
LIN {X 0,Y 86.923,Z 517.896,A -85,B 0,C 180,E1 -27652.581,E2 -27652.581} C_VEL
LIN {X 0,Y 92.05,Z 509.284,A -85,B 0,C 180,E1 -27658.498,E2 -27658.498} C_VEL
LIN {X 0,Y 96.963,Z 500.447,A -85,B 0,C 180,E1 -27662.926,E2 -27662.926} C_VEL
LIN {X 0,Y 101.93,Z 490.718,A -85,B 0,C 180,E1 -27666.486,E2 -27666.486} C_VEL
LIN {X 0,Y 106.637,Z 480.056,A -85,B 0,C 180,E1 -27669.367,E2 -27669.367} C_VEL
LIN {X 0,Y 110.724,Z 468.197,A -85,B 0,C 180,E1 -27671.791,E2 -27671.791} C_VEL
LIN {X 0,Y 114.003,Z 456.011,A -85,B 0,C 180,E1 -27673.568,E2 -27673.568} C_VEL
LIN {X 0,Y 116.538,Z 442.78,A -85,B 0,C 180,E1 -27674.877,E2 -27674.877} C_VEL
LIN {X 0,Y 118.155,Z 428.183,A -85,B 0,C 180,E1 -27675.691,E2 -27675.691} C_VEL
LIN {X 0,Y 120.393,Z 402.425,A -85,B 0,C 180,E1 -27676.804,E2 -27676.804} C_VEL
LIN {X 0,Y 116.398,Z 393.492,A -85,B 0,C 180,E1 -27680.454,E2 -27680.454} C_VEL
LIN {X 0,Y 112.096,Z 385.459,A -85,B 0,C 180,E1 -27684.969,E2 -27684.969} C_VEL
LIN {X 0,Y 109.402,Z 381.121,A -85,B 0,C 180,E1 -27688.257,E2 -27688.257} C_VEL
LIN {X 0,Y 107.358,Z 377.887,A -85,B 0,C 180,E1 -27691.148,E2 -27691.148} C_VEL
LIN {X 0,Y 105.047,Z 374.267,A -85,B 0,C 180,E1 -27695.054,E2 -27695.054} C_VEL
LIN {X 0,Y 102.752,Z 371.229,A -85,B 0,C 180,E1 -27700.001,E2 -27700.001} C_VEL
LIN {X 0,Y 102.154,Z 369.635,A -85,B 0,C 180,E1 -27701.905,E2 -27701.905} C_VEL
LIN {X 0,Y 100.129,Z 367.644,A -85,B 0,C 180,E1 -27711.929,E2 -27711.929} C_VEL
LIN {X 0,Y 100.395,Z 367.456,A -85,B 0,C 180,E1 -27718.996,E2 -27718.996} C_VEL
LIN {X 0,Y 102.367,Z 369.67,A -85,B 0,C 180,E1 -27727.271,E2 -27727.271} C_VEL
LIN {X 0,Y 104.245,Z 373.272,A -85,B 0,C 180,E1 -27732.038,E2 -27732.038} C_VEL
LIN {X 0,Y 105.46,Z 374.648,A -85,B 0,C 180,E1 -27734.286,E2 -27734.286} C_VEL
LIN {X 0,Y 108.278,Z 379.157,A -85,B 0,C 180,E1 -27738.808,E2 -27738.808} C_VEL
LIN {X 0,Y 111.13,Z 383.893,A -85,B 0,C 180,E1 -27742.544,E2 -27742.544} C_VEL
LIN {X 0,Y 114.926,Z 390.628,A -85,B 0,C 180,E1 -27746.715,E2 -27746.715} C_VEL
LIN {X 0,Y 117.552,Z 396.258,A -85,B 0,C 180,E1 -27749.307,E2 -27749.307} C_VEL
LIN {X 0,Y 119.944,Z 404.074,A -85,B 0,C 180,E1 -27751.702,E2 -27751.702} C_VEL
LIN {X 0,Y 120.227,Z 405.177,A -85,B 0,C 180,E1 -27751.988,E2 -27751.988} C_VEL
LIN {X 0,Y 116.87,Z 443.037,A -85,B 0,C 180,E1 -27753.771,E2 -27753.771} C_VEL
LIN {X 0,Y 114.505,Z 456.717,A -85,B 0,C 180,E1 -27754.914,E2 -27754.914} C_VEL
LIN {X 0,Y 111.297,Z 468.855,A -85,B 0,C 180,E1 -27756.384,E2 -27756.384} C_VEL
LIN {X 0,Y 107.471,Z 479.986,A -85,B 0,C 180,E1 -27758.309,E2 -27758.309} C_VEL
LIN {X 0,Y 103.247,Z 490.306,A -85,B 0,C 180,E1 -27760.78,E2 -27760.78} C_VEL
LIN {X 0,Y 98.125,Z 500.991,A -85,B 0,C 180,E1 -27764.261,E2 -27764.261} C_VEL
LIN {X 0,Y 92.977,Z 510.619,A -85,B 0,C 180,E1 -27768.599,E2 -27768.599} C_VEL
LIN {X 0,Y 88.538,Z 518.496,A -85,B 0,C 180,E1 -27773.468,E2 -27773.468} C_VEL
LIN {X 0,Y 83.898,Z 526.154,A -85,B 0,C 180,E1 -27779.831,E2 -27779.831} C_VEL
LIN {X 0,Y 80.251,Z 532.294,A -85,B 0,C 180,E1 -27786.795,E2 -27786.795} C_VEL
LIN {X 0,Y 78.016,Z 537.161,A -85,B 0,C 180,E1 -27794.325,E2 -27794.325} C_VEL
LIN {X 0,Y 76.924,Z 540.875,A -85,B 0,C 180,E1 -27802.127,E2 -27802.127} C_VEL
LIN {X 0,Y 76.851,Z 543.543,A -85,B 0,C 180,E1 -27810.004,E2 -27810.004} C_VEL
LIN {X 0,Y 76.784,Z 544.765,A -85,B 0,C 180,E1 -27815.255,E2 -27815.255} C_VEL
LIN {X 0,Y 77.203,Z 545.59,A -85,B 0,C 180,E1 -27820.494,E2 -27820.494} C_VEL
LIN {X 0,Y 79.637,Z 546,A -85,B 0,C 180,E1 -27830.675,E2 -27830.675} C_VEL
LIN {X 0,Y 84.369,Z 544.899,A -85,B 0,C 180,E1 -27839.991,E2 -27839.991} C_VEL
LIN {X 0,Y 87.557,Z 543.752,A -85,B 0,C 180,E1 -27844.189,E2 -27844.189} C_VEL
LIN {X 0,Y 91.122,Z 542.181,A -85,B 0,C 180,E1 -27848.102,E2 -27848.102} C_VEL
LIN {X 0,Y 97.308,Z 539.054,A -85,B 0,C 180,E1 -27853.328,E2 -27853.328} C_VEL
LIN {X 0,Y 104.091,Z 534.896,A -85,B 0,C 180,E1 -27857.965,E2 -27857.965} C_VEL
LIN {X 0,Y 112.795,Z 528.586,A -85,B 0,C 180,E1 -27862.604,E2 -27862.604} C_VEL
LIN {X 0,Y 120.882,Z 521.734,A -85,B 0,C 180,E1 -27865.947,E2 -27865.947} C_VEL
LIN {X 0,Y 129.394,Z 513.19,A -85,B 0,C 180,E1 -27868.814,E2 -27868.814} C_VEL
LIN {X 0,Y 136.7,Z 504.442,A -85,B 0,C 180,E1 -27870.931,E2 -27870.931} C_VEL
LIN {X 0,Y 144.121,Z 493.708,A -85,B 0,C 180,E1 -27872.871,E2 -27872.871} C_VEL
LIN {X 0,Y 150.279,Z 482.95,A -85,B 0,C 180,E1 -27874.194,E2 -27874.194} C_VEL
LIN {X 0,Y 155.779,Z 470.746,A -85,B 0,C 180,E1 -27875.287,E2 -27875.287} C_VEL
LIN {X 0,Y 159.873,Z 458.841,A -85,B 0,C 180,E1 -27876.047,E2 -27876.047} C_VEL
LIN {X 0,Y 162.984,Z 445.933,A -85,B 0,C 180,E1 -27876.63,E2 -27876.63} C_VEL
LIN {X 0,Y 163.675,Z 441.548,A -85,B 0,C 180,E1 -27876.844,E2 -27876.844} C_VEL
LIN {X 0,Y 161.915,Z 434.943,A -85,B 0,C 180,E1 -27880.178,E2 -27880.178} C_VEL
LIN {X 0,Y 160.705,Z 431.336,A -85,B 0,C 180,E1 -27882.665,E2 -27882.665} C_VEL
LIN {X 0,Y 159.433,Z 428.461,A -85,B 0,C 180,E1 -27885.791,E2 -27885.791} C_VEL
LIN {X 0,Y 158.225,Z 425.003,A -85,B 0,C 180,E1 -27891.057,E2 -27891.057} C_VEL
LIN {X 0,Y 157.954,Z 424.838,A -85,B 0,C 180,E1 -27893.379,E2 -27893.379} C_VEL
LIN {X 0,Y 157.834,Z 425.567,A -85,B 0,C 180,E1 -27895.503,E2 -27895.503} C_VEL
LIN {X 0,Y 157.787,Z 427.461,A -85,B 0,C 180,E1 -27897.55,E2 -27897.55} C_VEL
LIN {X 0,Y 158.059,Z 432.808,A -85,B 0,C 180,E1 -27901.494,E2 -27901.494} C_VEL
LIN {X 0,Y 158.667,Z 436.04,A -85,B 0,C 180,E1 -27904.177,E2 -27904.177} C_VEL
LIN {X 0,Y 159.853,Z 439.385,A -85,B 0,C 180,E1 -27907.342,E2 -27907.342} C_VEL
LIN {X 0,Y 161.137,Z 443.214,A -85,B 0,C 180,E1 -27910.254,E2 -27910.254} C_VEL
LIN {X 0,Y 157.889,Z 456.401,A -85,B 0,C 180,E1 -27910.839,E2 -27910.839} C_VEL
LIN {X 0,Y 153.893,Z 467.974,A -85,B 0,C 180,E1 -27911.64,E2 -27911.64} C_VEL
LIN {X 0,Y 148.614,Z 479.665,A -85,B 0,C 180,E1 -27912.739,E2 -27912.739} C_VEL
LIN {X 0,Y 142.553,Z 490.342,A -85,B 0,C 180,E1 -27914.116,E2 -27914.116} C_VEL
LIN {X 0,Y 135.228,Z 500.78,A -85,B 0,C 180,E1 -27915.95,E2 -27915.95} C_VEL
LIN {X 0,Y 127.54,Z 509.831,A -85,B 0,C 180,E1 -27918.089,E2 -27918.089} C_VEL
LIN {X 0,Y 118.743,Z 518.456,A -85,B 0,C 180,E1 -27920.951,E2 -27920.951} C_VEL
LIN {X 0,Y 109.986,Z 525.554,A -85,B 0,C 180,E1 -27924.411,E2 -27924.411} C_VEL
LIN {X 0,Y 100.869,Z 531.698,A -85,B 0,C 180,E1 -27928.918,E2 -27928.918} C_VEL
LIN {X 0,Y 93.062,Z 536.001,A -85,B 0,C 180,E1 -27933.823,E2 -27933.823} C_VEL
LIN {X 0,Y 88.485,Z 538.102,A -85,B 0,C 180,E1 -27937.41,E2 -27937.41} C_VEL
LIN {X 0,Y 83.274,Z 540.13,A -85,B 0,C 180,E1 -27942.469,E2 -27942.469} C_VEL
LIN {X 0,Y 77.201,Z 541.78,A -85,B 0,C 180,E1 -27950.409,E2 -27950.409} C_VEL
LIN {X 0,Y 72.288,Z 542.102,A -85,B 0,C 180,E1 -27960.911,E2 -27960.911} C_VEL
LIN {X 0,Y 70.68,Z 541.673,A -85,B 0,C 180,E1 -27966.559,E2 -27966.559} C_VEL
LIN {X 0,Y 69.648,Z 540.804,A -85,B 0,C 180,E1 -27972.375,E2 -27972.375} C_VEL
LIN {X 0,Y 69.265,Z 539.517,A -85,B 0,C 180,E1 -27978.287,E2 -27978.287} C_VEL
LIN {X 0,Y 70.284,Z 535.881,A -85,B 0,C 180,E1 -27989.549,E2 -27989.549} C_VEL
LIN {X 0,Y 72.216,Z 531.629,A -85,B 0,C 180,E1 -27998.39,E2 -27998.39} C_VEL
LIN {X 0,Y 75.976,Z 525.386,A -85,B 0,C 180,E1 -28007.491,E2 -28007.491} C_VEL
LIN {X 0,Y 80.41,Z 518.6,A -85,B 0,C 180,E1 -28014.525,E2 -28014.525} C_VEL
LIN {X 0,Y 85.869,Z 510.152,A -85,B 0,C 180,E1 -28020.762,E2 -28020.762} C_VEL
LIN {X 0,Y 91.096,Z 501.445,A -85,B 0,C 180,E1 -28025.349,E2 -28025.349} C_VEL
LIN {X 0,Y 96.92,Z 490.703,A -85,B 0,C 180,E1 -28029.378,E2 -28029.378} C_VEL
LIN {X 0,Y 101.282,Z 481.42,A -85,B 0,C 180,E1 -28031.899,E2 -28031.899} C_VEL
LIN {X 0,Y 105.582,Z 469.994,A -85,B 0,C 180,E1 -28034.336,E2 -28034.336} C_VEL
LIN {X 0,Y 109.32,Z 457.057,A -85,B 0,C 180,E1 -28036.276,E2 -28036.276} C_VEL
LIN {X 0,Y 112.033,Z 443.861,A -85,B 0,C 180,E1 -28037.612,E2 -28037.612} C_VEL
LIN {X 0,Y 113.726,Z 430.2,A -85,B 0,C 180,E1 -28038.398,E2 -28038.398} C_VEL
LIN {X 0,Y 116.018,Z 405.091,A -85,B 0,C 180,E1 -28039.467,E2 -28039.467} C_VEL
LIN {X 0,Y 112.775,Z 397.712,A -85,B 0,C 180,E1 -28042.829,E2 -28042.829} C_VEL
LIN {X 0,Y 109.321,Z 390.835,A -85,B 0,C 180,E1 -28046.932,E2 -28046.932} C_VEL
LIN {X 0,Y 105.799,Z 384.666,A -85,B 0,C 180,E1 -28051.986,E2 -28051.986} C_VEL
LIN {X 0,Y 103.259,Z 380.693,A -85,B 0,C 180,E1 -28056.627,E2 -28056.627} C_VEL
LIN {X 0,Y 101.268,Z 377.558,A -85,B 0,C 180,E1 -28061.599,E2 -28061.599} C_VEL
LIN {X 0,Y 100.852,Z 376.463,A -85,B 0,C 180,E1 -28063.1,E2 -28063.1} C_VEL
LIN {X 0,Y 99.224,Z 374.641,A -85,B 0,C 180,E1 -28072.547,E2 -28072.547} C_VEL
LIN {X 0,Y 99.515,Z 374.534,A -85,B 0,C 180,E1 -28078.988,E2 -28078.988} C_VEL
LIN {X 0,Y 101.096,Z 376.518,A -85,B 0,C 180,E1 -28086.235,E2 -28086.235} C_VEL
LIN {X 0,Y 102.95,Z 380.131,A -85,B 0,C 180,E1 -28091.318,E2 -28091.318} C_VEL
LIN {X 0,Y 103.966,Z 381.547,A -85,B 0,C 180,E1 -28093.374,E2 -28093.374} C_VEL
LIN {X 0,Y 106.342,Z 385.616,A -85,B 0,C 180,E1 -28097.512,E2 -28097.512} C_VEL
LIN {X 0,Y 109.022,Z 390.317,A -85,B 0,C 180,E1 -28101.322,E2 -28101.322} C_VEL
LIN {X 0,Y 112.245,Z 396.604,A -85,B 0,C 180,E1 -28105.21,E2 -28105.21} C_VEL
LIN {X 0,Y 114.132,Z 400.982,A -85,B 0,C 180,E1 -28107.288,E2 -28107.288} C_VEL
LIN {X 0,Y 115.91,Z 407.281,A -85,B 0,C 180,E1 -28109.32,E2 -28109.32} C_VEL
LIN {X 0,Y 112.565,Z 442.827,A -85,B 0,C 180,E1 -28110.969,E2 -28110.969} C_VEL
LIN {X 0,Y 110.004,Z 456.811,A -85,B 0,C 180,E1 -28112.112,E2 -28112.112} C_VEL
LIN {X 0,Y 106.544,Z 469.222,A -85,B 0,C 180,E1 -28113.619,E2 -28113.619} C_VEL
LIN {X 0,Y 101.927,Z 481.837,A -85,B 0,C 180,E1 -28115.893,E2 -28115.893} C_VEL
LIN {X 0,Y 96.898,Z 493.084,A -85,B 0,C 180,E1 -28118.773,E2 -28118.773} C_VEL
LIN {X 0,Y 92.094,Z 502.162,A -85,B 0,C 180,E1 -28121.928,E2 -28121.928} C_VEL
LIN {X 0,Y 86.518,Z 511.82,A -85,B 0,C 180,E1 -28126.659,E2 -28126.659} C_VEL
LIN {X 0,Y 81.091,Z 520.545,A -85,B 0,C 180,E1 -28132.655,E2 -28132.655} C_VEL
LIN {X 0,Y 76.349,Z 527.802,A -85,B 0,C 180,E1 -28139.588,E2 -28139.588} C_VEL
LIN {X 0,Y 72.727,Z 533.568,A -85,B 0,C 180,E1 -28147.265,E2 -28147.265} C_VEL
LIN {X 0,Y 70.604,Z 538.104,A -85,B 0,C 180,E1 -28155.595,E2 -28155.595} C_VEL
LIN {X 0,Y 69.728,Z 541.527,A -85,B 0,C 180,E1 -28164.22,E2 -28164.22} C_VEL
LIN {X 0,Y 69.749,Z 543.213,A -85,B 0,C 180,E1 -28170.004,E2 -28170.004} C_VEL
LIN {X 0,Y 69.727,Z 544.465,A -85,B 0,C 180,E1 -28175.789,E2 -28175.789} C_VEL
LIN {X 0,Y 70.213,Z 545.322,A -85,B 0,C 180,E1 -28181.552,E2 -28181.552} C_VEL
LIN {X 0,Y 71.303,Z 545.774,A -85,B 0,C 180,E1 -28187.203,E2 -28187.203} C_VEL
LIN {X 0,Y 75.307,Z 545.48,A -85,B 0,C 180,E1 -28197.819,E2 -28197.819} C_VEL
LIN {X 0,Y 81.764,Z 543.678,A -85,B 0,C 180,E1 -28206.995,E2 -28206.995} C_VEL
LIN {X 0,Y 85.641,Z 542.144,A -85,B 0,C 180,E1 -28211.038,E2 -28211.038} C_VEL
LIN {X 0,Y 93.264,Z 538.529,A -85,B 0,C 180,E1 -28217.103,E2 -28217.103} C_VEL
LIN {X 0,Y 102.015,Z 533.375,A -85,B 0,C 180,E1 -28222.401,E2 -28222.401} C_VEL
LIN {X 0,Y 110.011,Z 527.744,A -85,B 0,C 180,E1 -28226.154,E2 -28226.154} C_VEL
LIN {X 0,Y 118.524,Z 520.715,A -85,B 0,C 180,E1 -28229.297,E2 -28229.297} C_VEL
LIN {X 0,Y 127.365,Z 511.956,A -85,B 0,C 180,E1 -28231.995,E2 -28231.995} C_VEL
LIN {X 0,Y 135.674,Z 502.035,A -85,B 0,C 180,E1 -28234.166,E2 -28234.166} C_VEL
LIN {X 0,Y 141.832,Z 493.184,A -85,B 0,C 180,E1 -28235.579,E2 -28235.579} C_VEL
LIN {X 0,Y 148.144,Z 482.321,A -85,B 0,C 180,E1 -28236.807,E2 -28236.807} C_VEL
LIN {X 0,Y 153.903,Z 469.676,A -85,B 0,C 180,E1 -28237.847,E2 -28237.847} C_VEL
LIN {X 0,Y 158.087,Z 457.47,A -85,B 0,C 180,E1 -28238.563,E2 -28238.563} C_VEL
LIN {X 0,Y 160.984,Z 445.203,A -85,B 0,C 180,E1 -28239.083,E2 -28239.083} C_VEL
LIN {X 0,Y 159.887,Z 439.773,A -85,B 0,C 180,E1 -28242.08,E2 -28242.08} C_VEL
LIN {X 0,Y 159.188,Z 437.627,A -85,B 0,C 180,E1 -28243.818,E2 -28243.818} C_VEL
LIN {X 0,Y 158.265,Z 435.207,A -85,B 0,C 180,E1 -28246.533,E2 -28246.533} C_VEL
LIN {X 0,Y 157.26,Z 431.988,A -85,B 0,C 180,E1 -28251.649,E2 -28251.649} C_VEL
LIN {X 0,Y 157.333,Z 431.784,A -85,B 0,C 180,E1 -28258.081,E2 -28258.081} C_VEL
LIN {X 0,Y 158.51,Z 435.505,A -85,B 0,C 180,E1 -28263.655,E2 -28263.655} C_VEL
LIN {X 0,Y 158.667,Z 436.04,A -85,B 0,C 180,E1 -28264.177,E2 -28264.177} C_VEL
LIN {X 0,Y 158.994,Z 438.064,A -85,B 0,C 180,E1 -28265.442,E2 -28265.442} C_VEL
LIN {X 0,Y 159.014,Z 441.062,A -85,B 0,C 180,E1 -28266.456,E2 -28266.456} C_VEL
LIN {X 0,Y 158.536,Z 445.95,A -85,B 0,C 180,E1 -28267.446,E2 -28267.446} C_VEL
LIN {X 0,Y 157.491,Z 451.344,A -85,B 0,C 180,E1 -28268.06,E2 -28268.06} C_VEL
LIN {X 0,Y 156.778,Z 454.101,A -85,B 0,C 180,E1 -28268.222,E2 -28268.222} C_VEL
LIN {X 0,Y 152.534,Z 466.734,A -85,B 0,C 180,E1 -28268.99,E2 -28268.99} C_VEL
LIN {X 0,Y 147.171,Z 478.581,A -85,B 0,C 180,E1 -28269.954,E2 -28269.954} C_VEL
LIN {X 0,Y 140.522,Z 490.226,A -85,B 0,C 180,E1 -28271.339,E2 -28271.339} C_VEL
LIN {X 0,Y 133.412,Z 500.193,A -85,B 0,C 180,E1 -28272.944,E2 -28272.944} C_VEL
LIN {X 0,Y 125.468,Z 509.37,A -85,B 0,C 180,E1 -28274.923,E2 -28274.923} C_VEL
LIN {X 0,Y 116.496,Z 517.993,A -85,B 0,C 180,E1 -28277.557,E2 -28277.557} C_VEL
LIN {X 0,Y 107.172,Z 525.337,A -85,B 0,C 180,E1 -28280.851,E2 -28280.851} C_VEL
LIN {X 0,Y 97.325,Z 531.687,A -85,B 0,C 180,E1 -28285.258,E2 -28285.258} C_VEL
LIN {X 0,Y 89.196,Z 535.944,A -85,B 0,C 180,E1 -28289.914,E2 -28289.914} C_VEL
LIN {X 0,Y 84.227,Z 538.117,A -85,B 0,C 180,E1 -28293.44,E2 -28293.44} C_VEL
LIN {X 0,Y 77.841,Z 540.407,A -85,B 0,C 180,E1 -28299.2,E2 -28299.2} C_VEL
LIN {X 0,Y 71.7,Z 541.927,A -85,B 0,C 180,E1 -28306.67,E2 -28306.67} C_VEL
LIN {X 0,Y 68.528,Z 542.327,A -85,B 0,C 180,E1 -28312.019,E2 -28312.019} C_VEL
LIN {X 0,Y 65.553,Z 542.283,A -85,B 0,C 180,E1 -28319.061,E2 -28319.061} C_VEL
LIN {X 0,Y 62.775,Z 541.124,A -85,B 0,C 180,E1 -28330.37,E2 -28330.37} C_VEL
LIN {X 0,Y 62.191,Z 539.872,A -85,B 0,C 180,E1 -28336.933,E2 -28336.933} C_VEL
LIN {X 0,Y 62.647,Z 537.225,A -85,B 0,C 180,E1 -28346.78,E2 -28346.78} C_VEL
LIN {X 0,Y 63.527,Z 535.305,A -85,B 0,C 180,E1 -28352.137,E2 -28352.137} C_VEL
LIN {X 0,Y 66.11,Z 530.541,A -85,B 0,C 180,E1 -28362.271,E2 -28362.271} C_VEL
LIN {X 0,Y 69.944,Z 524.988,A -85,B 0,C 180,E1 -28370.585,E2 -28370.585} C_VEL
LIN {X 0,Y 74.923,Z 518.067,A -85,B 0,C 180,E1 -28377.965,E2 -28377.965} C_VEL
LIN {X 0,Y 80.939,Z 509.385,A -85,B 0,C 180,E1 -28384.356,E2 -28384.356} C_VEL
LIN {X 0,Y 86.586,Z 500.489,A -85,B 0,C 180,E1 -28388.975,E2 -28388.975} C_VEL
LIN {X 0,Y 92.184,Z 490.687,A -85,B 0,C 180,E1 -28392.575,E2 -28392.575} C_VEL
LIN {X 0,Y 96.78,Z 481.359,A -85,B 0,C 180,E1 -28395.07,E2 -28395.07} C_VEL
LIN {X 0,Y 101.317,Z 469.846,A -85,B 0,C 180,E1 -28397.473,E2 -28397.473} C_VEL
LIN {X 0,Y 105.199,Z 456.932,A -85,B 0,C 180,E1 -28399.366,E2 -28399.366} C_VEL
LIN {X 0,Y 107.918,Z 444.28,A -85,B 0,C 180,E1 -28400.619,E2 -28400.619} C_VEL
LIN {X 0,Y 109.726,Z 430.556,A -85,B 0,C 180,E1 -28401.39,E2 -28401.39} C_VEL
LIN {X 0,Y 111.841,Z 407.803,A -85,B 0,C 180,E1 -28402.387,E2 -28402.387} C_VEL
LIN {X 0,Y 108.832,Z 400.735,A -85,B 0,C 180,E1 -28406.035,E2 -28406.035} C_VEL
LIN {X 0,Y 105.674,Z 394.253,A -85,B 0,C 180,E1 -28410.496,E2 -28410.496} C_VEL
LIN {X 0,Y 103.285,Z 390.069,A -85,B 0,C 180,E1 -28414.564,E2 -28414.564} C_VEL
LIN {X 0,Y 101.636,Z 387.183,A -85,B 0,C 180,E1 -28418.073,E2 -28418.073} C_VEL
LIN {X 0,Y 99.81,Z 383.757,A -85,B 0,C 180,E1 -28423.46,E2 -28423.46} C_VEL
LIN {X 0,Y 99.397,Z 383.19,A -85,B 0,C 180,E1 -28425.05,E2 -28425.05} C_VEL
LIN {X 0,Y 98.354,Z 381.702,A -85,B 0,C 180,E1 -28432.481,E2 -28432.481} C_VEL
LIN {X 0,Y 98.479,Z 381.499,A -85,B 0,C 180,E1 -28437.511,E2 -28437.511} C_VEL
LIN {X 0,Y 99.908,Z 383.477,A -85,B 0,C 180,E1 -28445.36,E2 -28445.36} C_VEL
LIN {X 0,Y 101.672,Z 386.995,A -85,B 0,C 180,E1 -28450.579,E2 -28450.579} C_VEL
LIN {X 0,Y 102.501,Z 388.436,A -85,B 0,C 180,E1 -28452.435,E2 -28452.435} C_VEL
LIN {X 0,Y 104.363,Z 391.861,A -85,B 0,C 180,E1 -28455.996,E2 -28455.996} C_VEL
LIN {X 0,Y 107.118,Z 397.066,A -85,B 0,C 180,E1 -28460.273,E2 -28460.273} C_VEL
LIN {X 0,Y 110.236,Z 403.899,A -85,B 0,C 180,E1 -28464.356,E2 -28464.356} C_VEL
LIN {X 0,Y 111.827,Z 409.361,A -85,B 0,C 180,E1 -28466.419,E2 -28466.419} C_VEL
LIN {X 0,Y 108.546,Z 442.544,A -85,B 0,C 180,E1 -28467.935,E2 -28467.935} C_VEL
LIN {X 0,Y 105.885,Z 456.498,A -85,B 0,C 180,E1 -28469.042,E2 -28469.042} C_VEL
LIN {X 0,Y 102.421,Z 468.577,A -85,B 0,C 180,E1 -28470.462,E2 -28470.462} C_VEL
LIN {X 0,Y 97.883,Z 480.475,A -85,B 0,C 180,E1 -28472.479,E2 -28472.479} C_VEL
LIN {X 0,Y 93.219,Z 490.634,A -85,B 0,C 180,E1 -28474.932,E2 -28474.932} C_VEL
LIN {X 0,Y 87.502,Z 501.194,A -85,B 0,C 180,E1 -28478.461,E2 -28478.461} C_VEL
LIN {X 0,Y 81.667,Z 510.693,A -85,B 0,C 180,E1 -28482.995,E2 -28482.995} C_VEL
LIN {X 0,Y 76.35,Z 518.7,A -85,B 0,C 180,E1 -28488.424,E2 -28488.424} C_VEL
LIN {X 0,Y 71.07,Z 526.07,A -85,B 0,C 180,E1 -28495.352,E2 -28495.352} C_VEL
LIN {X 0,Y 66.182,Z 533.063,A -85,B 0,C 180,E1 -28504.869,E2 -28504.869} C_VEL
LIN {X 0,Y 63.727,Z 537.674,A -85,B 0,C 180,E1 -28514.001,E2 -28514.001} C_VEL
LIN {X 0,Y 62.649,Z 541.156,A -85,B 0,C 180,E1 -28523.564,E2 -28523.564} C_VEL
LIN {X 0,Y 62.67,Z 542.884,A -85,B 0,C 180,E1 -28530.005,E2 -28530.005} C_VEL
LIN {X 0,Y 62.654,Z 544.164,A -85,B 0,C 180,E1 -28536.445,E2 -28536.445} C_VEL
LIN {X 0,Y 63.264,Z 545.051,A -85,B 0,C 180,E1 -28542.842,E2 -28542.842} C_VEL
LIN {X 0,Y 64.534,Z 545.551,A -85,B 0,C 180,E1 -28549.074,E2 -28549.074} C_VEL
LIN {X 0,Y 69.082,Z 545.324,A -85,B 0,C 180,E1 -28560.58,E2 -28560.58} C_VEL
LIN {X 0,Y 76.186,Z 543.588,A -85,B 0,C 180,E1 -28570.225,E2 -28570.225} C_VEL
LIN {X 0,Y 80.416,Z 542.106,A -85,B 0,C 180,E1 -28574.364,E2 -28574.364} C_VEL
LIN {X 0,Y 89.603,Z 538.042,A -85,B 0,C 180,E1 -28581.136,E2 -28581.136} C_VEL
LIN {X 0,Y 97.839,Z 533.468,A -85,B 0,C 180,E1 -28585.702,E2 -28585.702} C_VEL
LIN {X 0,Y 106.224,Z 527.912,A -85,B 0,C 180,E1 -28589.333,E2 -28589.333} C_VEL
LIN {X 0,Y 115.074,Z 520.999,A -85,B 0,C 180,E1 -28592.326,E2 -28592.326} C_VEL
LIN {X 0,Y 124.201,Z 512.361,A -85,B 0,C 180,E1 -28594.878,E2 -28594.878} C_VEL
LIN {X 0,Y 131.957,Z 503.54,A -85,B 0,C 180,E1 -28596.746,E2 -28596.746} C_VEL
LIN {X 0,Y 139.062,Z 493.869,A -85,B 0,C 180,E1 -28598.229,E2 -28598.229} C_VEL
LIN {X 0,Y 145.514,Z 483.28,A -85,B 0,C 180,E1 -28599.357,E2 -28599.357} C_VEL
LIN {X 0,Y 151.448,Z 470.829,A -85,B 0,C 180,E1 -28600.323,E2 -28600.323} C_VEL
LIN {X 0,Y 156.061,Z 457.934,A -85,B 0,C 180,E1 -28601.037,E2 -28601.037} C_VEL
LIN {X 0,Y 158.409,Z 448.849,A -85,B 0,C 180,E1 -28601.425,E2 -28601.425} C_VEL
LIN {X 0,Y 157.759,Z 444.583,A -85,B 0,C 180,E1 -28604.166,E2 -28604.166} C_VEL
LIN {X 0,Y 156.907,Z 441.903,A -85,B 0,C 180,E1 -28607.253,E2 -28607.253} C_VEL
LIN {X 0,Y 156.207,Z 438.959,A -85,B 0,C 180,E1 -28612.243,E2 -28612.243} C_VEL
LIN {X 0,Y 156.328,Z 438.911,A -85,B 0,C 180,E1 -28618.068,E2 -28618.068} C_VEL
LIN {X 0,Y 157.08,Z 442.295,A -85,B 0,C 180,E1 -28623.046,E2 -28623.046} C_VEL
LIN {X 0,Y 157.997,Z 445.9,A -85,B 0,C 180,E1 -28626.546,E2 -28626.546} C_VEL
LIN {X 0,Y 158.445,Z 447.491,A -85,B 0,C 180,E1 -28627.922,E2 -28627.922} C_VEL
LIN {X 0,Y 156.778,Z 454.101,A -85,B 0,C 180,E1 -28628.222,E2 -28628.222} C_VEL
LIN {X 0,Y 154.964,Z 459.732,A -85,B 0,C 180,E1 -28628.265,E2 -28628.265} C_VEL
LIN {X 0,Y 151.001,Z 468.743,A -85,B 0,C 180,E1 -28627.795,E2 -28627.795} C_VEL
LIN {X 0,Y 146.342,Z 477.414,A -85,B 0,C 180,E1 -28627.412,E2 -28627.412} C_VEL
LIN {X 0,Y 143.42,Z 482.506,A -85,B 0,C 180,E1 -28627.623,E2 -28627.623} C_VEL
LIN {X 0,Y 136.936,Z 492.874,A -85,B 0,C 180,E1 -28628.858,E2 -28628.858} C_VEL
LIN {X 0,Y 130.329,Z 501.599,A -85,B 0,C 180,E1 -28630.212,E2 -28630.212} C_VEL
LIN {X 0,Y 122.174,Z 510.573,A -85,B 0,C 180,E1 -28632.055,E2 -28632.055} C_VEL
LIN {X 0,Y 113.647,Z 518.396,A -85,B 0,C 180,E1 -28634.322,E2 -28634.322} C_VEL
LIN {X 0,Y 104.8,Z 525.133,A -85,B 0,C 180,E1 -28637.127,E2 -28637.127} C_VEL
LIN {X 0,Y 97.235,Z 529.981,A -85,B 0,C 180,E1 -28640.005,E2 -28640.005} C_VEL
LIN {X 0,Y 88.562,Z 534.628,A -85,B 0,C 180,E1 -28644.126,E2 -28644.126} C_VEL
LIN {X 0,Y 80.425,Z 538.129,A -85,B 0,C 180,E1 -28649.084,E2 -28649.084} C_VEL
LIN {X 0,Y 72.712,Z 540.676,A -85,B 0,C 180,E1 -28655.447,E2 -28655.447} C_VEL
LIN {X 0,Y 66.565,Z 542.052,A -85,B 0,C 180,E1 -28662.342,E2 -28662.342} C_VEL
LIN {X 0,Y 62.927,Z 542.514,A -85,B 0,C 180,E1 -28667.919,E2 -28667.919} C_VEL
LIN {X 0,Y 59.004,Z 542.473,A -85,B 0,C 180,E1 -28676.491,E2 -28676.491} C_VEL
LIN {X 0,Y 56.003,Z 541.426,A -85,B 0,C 180,E1 -28687.879,E2 -28687.879} C_VEL
LIN {X 0,Y 55.176,Z 540.225,A -85,B 0,C 180,E1 -28695.236,E2 -28695.236} C_VEL
LIN {X 0,Y 55.459,Z 537.647,A -85,B 0,C 180,E1 -28706.362,E2 -28706.362} C_VEL
LIN {X 0,Y 56.556,Z 535.401,A -85,B 0,C 180,E1 -28713.425,E2 -28713.425} C_VEL
LIN {X 0,Y 59.191,Z 531.071,A -85,B 0,C 180,E1 -28723.732,E2 -28723.732} C_VEL
LIN {X 0,Y 64.159,Z 524.589,A -85,B 0,C 180,E1 -28734.249,E2 -28734.249} C_VEL
LIN {X 0,Y 69.743,Z 517.482,A -85,B 0,C 180,E1 -28741.935,E2 -28741.935} C_VEL
LIN {X 0,Y 76.352,Z 508.62,A -85,B 0,C 180,E1 -28748.407,E2 -28748.407} C_VEL
LIN {X 0,Y 82.483,Z 499.529,A -85,B 0,C 180,E1 -28752.967,E2 -28752.967} C_VEL
LIN {X 0,Y 88.534,Z 489.424,A -85,B 0,C 180,E1 -28756.41,E2 -28756.41} C_VEL
LIN {X 0,Y 93.948,Z 478.241,A -85,B 0,C 180,E1 -28759.232,E2 -28759.232} C_VEL
LIN {X 0,Y 98.765,Z 465.729,A -85,B 0,C 180,E1 -28761.507,E2 -28761.507} C_VEL
LIN {X 0,Y 102.416,Z 452.961,A -85,B 0,C 180,E1 -28763.087,E2 -28763.087} C_VEL
LIN {X 0,Y 104.91,Z 439.915,A -85,B 0,C 180,E1 -28764.18,E2 -28764.18} C_VEL
LIN {X 0,Y 108.026,Z 410.764,A -85,B 0,C 180,E1 -28765.441,E2 -28765.441} C_VEL
LIN {X 0,Y 105.256,Z 404.067,A -85,B 0,C 180,E1 -28769.391,E2 -28769.391} C_VEL
LIN {X 0,Y 102.939,Z 399.184,A -85,B 0,C 180,E1 -28773.273,E2 -28773.273} C_VEL
LIN {X 0,Y 101.25,Z 395.871,A -85,B 0,C 180,E1 -28776.692,E2 -28776.692} C_VEL
LIN {X 0,Y 100.121,Z 393.75,A -85,B 0,C 180,E1 -28779.452,E2 -28779.452} C_VEL
LIN {X 0,Y 98.543,Z 390.287,A -85,B 0,C 180,E1 -28784.917,E2 -28784.917} C_VEL
LIN {X 0,Y 97.463,Z 388.707,A -85,B 0,C 180,E1 -28793.003,E2 -28793.003} C_VEL
LIN {X 0,Y 97.602,Z 388.554,A -85,B 0,C 180,E1 -28797.489,E2 -28797.489} C_VEL
LIN {X 0,Y 98.706,Z 390.274,A -85,B 0,C 180,E1 -28804.274,E2 -28804.274} C_VEL
LIN {X 0,Y 100.309,Z 393.738,A -85,B 0,C 180,E1 -28809.578,E2 -28809.578} C_VEL
LIN {X 0,Y 102.376,Z 397.881,A -85,B 0,C 180,E1 -28814.25,E2 -28814.25} C_VEL
LIN {X 0,Y 104.882,Z 403.165,A -85,B 0,C 180,E1 -28818.642,E2 -28818.642} C_VEL
LIN {X 0,Y 107.463,Z 409.335,A -85,B 0,C 180,E1 -28822.436,E2 -28822.436} C_VEL
LIN {X 0,Y 108.034,Z 411.613,A -85,B 0,C 180,E1 -28823.316,E2 -28823.316} C_VEL
LIN {X 0,Y 104.776,Z 442.807,A -85,B 0,C 180,E1 -28824.718,E2 -28824.718} C_VEL
LIN {X 0,Y 102.033,Z 456.459,A -85,B 0,C 180,E1 -28825.763,E2 -28825.763} C_VEL
LIN {X 0,Y 98.261,Z 468.939,A -85,B 0,C 180,E1 -28827.187,E2 -28827.187} C_VEL
LIN {X 0,Y 93.527,Z 480.72,A -85,B 0,C 180,E1 -28829.134,E2 -28829.134} C_VEL
LIN {X 0,Y 88.626,Z 490.797,A -85,B 0,C 180,E1 -28831.526,E2 -28831.526} C_VEL
LIN {X 0,Y 82.591,Z 501.296,A -85,B 0,C 180,E1 -28835.019,E2 -28835.019} C_VEL
LIN {X 0,Y 76.972,Z 509.876,A -85,B 0,C 180,E1 -28839.102,E2 -28839.102} C_VEL
LIN {X 0,Y 71.389,Z 517.603,A -85,B 0,C 180,E1 -28844.229,E2 -28844.229} C_VEL
LIN {X 0,Y 65.304,Z 525.463,A -85,B 0,C 180,E1 -28851.777,E2 -28851.777} C_VEL
LIN {X 0,Y 59.786,Z 532.537,A -85,B 0,C 180,E1 -28861.958,E2 -28861.958} C_VEL
LIN {X 0,Y 56.904,Z 537.226,A -85,B 0,C 180,E1 -28872.021,E2 -28872.021} C_VEL
LIN {X 0,Y 55.589,Z 540.769,A -85,B 0,C 180,E1 -28882.742,E2 -28882.742} C_VEL
LIN {X 0,Y 55.579,Z 542.554,A -85,B 0,C 180,E1 -28890.005,E2 -28890.005} C_VEL
LIN {X 0,Y 55.593,Z 543.863,A -85,B 0,C 180,E1 -28897.268,E2 -28897.268} C_VEL
LIN {X 0,Y 57.858,Z 545.312,A -85,B 0,C 180,E1 -28911.377,E2 -28911.377} C_VEL
LIN {X 0,Y 60.103,Z 545.445,A -85,B 0,C 180,E1 -28917.892,E2 -28917.892} C_VEL
LIN {X 0,Y 66.719,Z 544.519,A -85,B 0,C 180,E1 -28929.204,E2 -28929.204} C_VEL
LIN {X 0,Y 75.501,Z 542.067,A -85,B 0,C 180,E1 -28938.137,E2 -28938.137} C_VEL
LIN {X 0,Y 84.665,Z 538.38,A -85,B 0,C 180,E1 -28944.475,E2 -28944.475} C_VEL
LIN {X 0,Y 94.024,Z 533.572,A -85,B 0,C 180,E1 -28949.275,E2 -28949.275} C_VEL
LIN {X 0,Y 102.792,Z 528.094,A -85,B 0,C 180,E1 -28952.73,E2 -28952.73} C_VEL
LIN {X 0,Y 111.955,Z 521.269,A -85,B 0,C 180,E1 -28955.544,E2 -28955.544} C_VEL
LIN {X 0,Y 121.366,Z 512.776,A -85,B 0,C 180,E1 -28957.903,E2 -28957.903} C_VEL
LIN {X 0,Y 129.334,Z 504.076,A -85,B 0,C 180,E1 -28959.618,E2 -28959.618} C_VEL
LIN {X 0,Y 136.601,Z 494.554,A -85,B 0,C 180,E1 -28960.98,E2 -28960.98} C_VEL
LIN {X 0,Y 143.177,Z 484.157,A -85,B 0,C 180,E1 -28962.002,E2 -28962.002} C_VEL
LIN {X 0,Y 149.242,Z 472.085,A -85,B 0,C 180,E1 -28962.869,E2 -28962.869} C_VEL
LIN {X 0,Y 153.921,Z 459.684,A -85,B 0,C 180,E1 -28963.512,E2 -28963.512} C_VEL
LIN {X 0,Y 155.95,Z 452.683,A -85,B 0,C 180,E1 -28963.831,E2 -28963.831} C_VEL
LIN {X 0,Y 155.706,Z 450.626,A -85,B 0,C 180,E1 -28965.46,E2 -28965.46} C_VEL
LIN {X 0,Y 155.229,Z 448.576,A -85,B 0,C 180,E1 -28967.913,E2 -28967.913} C_VEL
LIN {X 0,Y 154.862,Z 445.943,A -85,B 0,C 180,E1 -28972.176,E2 -28972.176} C_VEL
LIN {X 0,Y 154.899,Z 445.843,A -85,B 0,C 180,E1 -28977.725,E2 -28977.725} C_VEL
LIN {X 0,Y 155.347,Z 449.119,A -85,B 0,C 180,E1 -28982.594,E2 -28982.594} C_VEL
LIN {X 0,Y 155.82,Z 452.07,A -85,B 0,C 180,E1 -28985.54,E2 -28985.54} C_VEL
LIN {X 0,Y 151.522,Z 465.399,A -85,B 0,C 180,E1 -28986.287,E2 -28986.287} C_VEL
LIN {X 0,Y 146.088,Z 477.504,A -85,B 0,C 180,E1 -28987.138,E2 -28987.138} C_VEL
LIN {X 0,Y 143.42,Z 482.506,A -85,B 0,C 180,E1 -28987.623,E2 -28987.623} C_VEL
LIN {X 0,Y 140.277,Z 487.565,A -85,B 0,C 180,E1 -28987.882,E2 -28987.882} C_VEL
LIN {X 0,Y 134.294,Z 495.482,A -85,B 0,C 180,E1 -28987.694,E2 -28987.694} C_VEL
LIN {X 0,Y 127.78,Z 502.898,A -85,B 0,C 180,E1 -28987.602,E2 -28987.602} C_VEL
LIN {X 0,Y 123.814,Z 507.111,A -85,B 0,C 180,E1 -28988.07,E2 -28988.07} C_VEL
LIN {X 0,Y 115.897,Z 514.795,A -85,B 0,C 180,E1 -28989.792,E2 -28989.792} C_VEL
LIN {X 0,Y 106.106,Z 522.65,A -85,B 0,C 180,E1 -28992.308,E2 -28992.308} C_VEL
LIN {X 0,Y 98.111,Z 527.98,A -85,B 0,C 180,E1 -28994.741,E2 -28994.741} C_VEL
LIN {X 0,Y 88.125,Z 533.443,A -85,B 0,C 180,E1 -28998.604,E2 -28998.604} C_VEL
LIN {X 0,Y 77.13,Z 538.122,A -85,B 0,C 180,E1 -29004.322,E2 -29004.322} C_VEL
LIN {X 0,Y 67.861,Z 540.958,A -85,B 0,C 180,E1 -29011.188,E2 -29011.188} C_VEL
LIN {X 0,Y 61.864,Z 542.176,A -85,B 0,C 180,E1 -29017.316,E2 -29017.316} C_VEL
LIN {X 0,Y 57.695,Z 542.696,A -85,B 0,C 180,E1 -29023.033,E2 -29023.033} C_VEL
LIN {X 0,Y 52.58,Z 542.661,A -85,B 0,C 180,E1 -29033.322,E2 -29033.322} C_VEL
LIN {X 0,Y 49.342,Z 541.712,A -85,B 0,C 180,E1 -29044.697,E2 -29044.697} C_VEL
LIN {X 0,Y 48.215,Z 540.576,A -85,B 0,C 180,E1 -29053.044,E2 -29053.044} C_VEL
LIN {X 0,Y 48.272,Z 538.063,A -85,B 0,C 180,E1 -29065.819,E2 -29065.819} C_VEL
LIN {X 0,Y 49.246,Z 536.276,A -85,B 0,C 180,E1 -29072.551,E2 -29072.551} C_VEL
LIN {X 0,Y 52.323,Z 531.597,A -85,B 0,C 180,E1 -29085.577,E2 -29085.577} C_VEL
LIN {X 0,Y 57.763,Z 525.197,A -85,B 0,C 180,E1 -29097.14,E2 -29097.14} C_VEL
LIN {X 0,Y 63.829,Z 518.224,A -85,B 0,C 180,E1 -29105.308,E2 -29105.308} C_VEL
LIN {X 0,Y 70.918,Z 509.478,A -85,B 0,C 180,E1 -29111.978,E2 -29111.978} C_VEL
LIN {X 0,Y 78.117,Z 499.537,A -85,B 0,C 180,E1 -29116.963,E2 -29116.963} C_VEL
LIN {X 0,Y 84.521,Z 489.367,A -85,B 0,C 180,E1 -29120.271,E2 -29120.271} C_VEL
LIN {X 0,Y 90.214,Z 478.127,A -85,B 0,C 180,E1 -29122.982,E2 -29122.982} C_VEL
LIN {X 0,Y 95.19,Z 465.709,A -85,B 0,C 180,E1 -29125.135,E2 -29125.135} C_VEL
LIN {X 0,Y 99.032,Z 452.741,A -85,B 0,C 180,E1 -29126.636,E2 -29126.636} C_VEL
LIN {X 0,Y 101.592,Z 439.784,A -85,B 0,C 180,E1 -29127.659,E2 -29127.659} C_VEL
LIN {X 0,Y 104.5,Z 413.87,A -85,B 0,C 180,E1 -29128.711,E2 -29128.711} C_VEL
LIN {X 0,Y 102.175,Z 407.921,A -85,B 0,C 180,E1 -29132.701,E2 -29132.701} C_VEL
LIN {X 0,Y 100.016,Z 403.014,A -85,B 0,C 180,E1 -29137.256,E2 -29137.256} C_VEL
LIN {X 0,Y 98.678,Z 400.308,A -85,B 0,C 180,E1 -29140.848,E2 -29140.848} C_VEL
LIN {X 0,Y 97.351,Z 397.08,A -85,B 0,C 180,E1 -29146.231,E2 -29146.231} C_VEL
LIN {X 0,Y 96.578,Z 395.654,A -85,B 0,C 180,E1 -29154.243,E2 -29154.243} C_VEL
LIN {X 0,Y 96.805,Z 395.793,A -85,B 0,C 180,E1 -29158.439,E2 -29158.439} C_VEL
LIN {X 0,Y 97.559,Z 397.167,A -85,B 0,C 180,E1 -29163.277,E2 -29163.277} C_VEL
LIN {X 0,Y 99.299,Z 401.261,A -85,B 0,C 180,E1 -29169.483,E2 -29169.483} C_VEL
LIN {X 0,Y 100.747,Z 404.59,A -85,B 0,C 180,E1 -29173.039,E2 -29173.039} C_VEL
LIN {X 0,Y 102.908,Z 409.684,A -85,B 0,C 180,E1 -29177.256,E2 -29177.256} C_VEL
LIN {X 0,Y 104.573,Z 414.089,A -85,B 0,C 180,E1 -29180.036,E2 -29180.036} C_VEL
LIN {X 0,Y 101.432,Z 442.55,A -85,B 0,C 180,E1 -29181.241,E2 -29181.241} C_VEL
LIN {X 0,Y 98.67,Z 455.874,A -85,B 0,C 180,E1 -29182.197,E2 -29182.197} C_VEL
LIN {X 0,Y 94.838,Z 468.28,A -85,B 0,C 180,E1 -29183.51,E2 -29183.51} C_VEL
LIN {X 0,Y 89.52,Z 480.952,A -85,B 0,C 180,E1 -29185.475,E2 -29185.475} C_VEL
LIN {X 0,Y 84.38,Z 490.951,A -85,B 0,C 180,E1 -29187.763,E2 -29187.763} C_VEL
LIN {X 0,Y 78.015,Z 501.391,A -85,B 0,C 180,E1 -29191.159,E2 -29191.159} C_VEL
LIN {X 0,Y 71.378,Z 510.753,A -85,B 0,C 180,E1 -29195.686,E2 -29195.686} C_VEL
LIN {X 0,Y 65.323,Z 518.461,A -85,B 0,C 180,E1 -29201.146,E2 -29201.146} C_VEL
LIN {X 0,Y 58.859,Z 525.986,A -85,B 0,C 180,E1 -29208.957,E2 -29208.957} C_VEL
LIN {X 0,Y 53.588,Z 532.008,A -85,B 0,C 180,E1 -29218.366,E2 -29218.366} C_VEL
LIN {X 0,Y 50.149,Z 536.766,A -85,B 0,C 180,E1 -29229.497,E2 -29229.497} C_VEL
LIN {X 0,Y 48.558,Z 540.379,A -85,B 0,C 180,E1 -29241.684,E2 -29241.684} C_VEL
LIN {X 0,Y 48.478,Z 542.221,A -85,B 0,C 180,E1 -29250.006,E2 -29250.006} C_VEL
LIN {X 0,Y 48.561,Z 543.563,A -85,B 0,C 180,E1 -29258.327,E2 -29258.327} C_VEL
LIN {X 0,Y 51.304,Z 545.069,A -85,B 0,C 180,E1 -29274.271,E2 -29274.271} C_VEL
LIN {X 0,Y 53.896,Z 545.249,A -85,B 0,C 180,E1 -29281.445,E2 -29281.445} C_VEL
LIN {X 0,Y 61.37,Z 544.395,A -85,B 0,C 180,E1 -29293.408,E2 -29293.408} C_VEL
LIN {X 0,Y 70.958,Z 542.016,A -85,B 0,C 180,E1 -29302.412,E2 -29302.412} C_VEL
LIN {X 0,Y 80.136,Z 538.685,A -85,B 0,C 180,E1 -29308.252,E2 -29308.252} C_VEL
LIN {X 0,Y 90.6,Z 533.678,A -85,B 0,C 180,E1 -29313.141,E2 -29313.141} C_VEL
LIN {X 0,Y 101.304,Z 527.269,A -85,B 0,C 180,E1 -29316.819,E2 -29316.819} C_VEL
LIN {X 0,Y 110.8,Z 520.289,A -85,B 0,C 180,E1 -29319.329,E2 -29319.329} C_VEL
LIN {X 0,Y 120.491,Z 511.574,A -85,B 0,C 180,E1 -29321.417,E2 -29321.417} C_VEL
LIN {X 0,Y 128.706,Z 502.666,A -85,B 0,C 180,E1 -29322.866,E2 -29322.866} C_VEL
LIN {X 0,Y 135.305,Z 494.069,A -85,B 0,C 180,E1 -29323.937,E2 -29323.937} C_VEL
LIN {X 0,Y 141.996,Z 483.611,A -85,B 0,C 180,E1 -29324.833,E2 -29324.833} C_VEL
LIN {X 0,Y 147.918,Z 471.98,A -85,B 0,C 180,E1 -29325.556,E2 -29325.556} C_VEL
LIN {X 0,Y 152.981,Z 458.643,A -85,B 0,C 180,E1 -29326.167,E2 -29326.167} C_VEL
LIN {X 0,Y 153.483,Z 456.85,A -85,B 0,C 180,E1 -29326.428,E2 -29326.428} C_VEL
LIN {X 0,Y 153.239,Z 455.26,A -85,B 0,C 180,E1 -29328.425,E2 -29328.425} C_VEL
LIN {X 0,Y 153.041,Z 452.801,A -85,B 0,C 180,E1 -29332.745,E2 -29332.745} C_VEL
LIN {X 0,Y 153.075,Z 452.812,A -85,B 0,C 180,E1 -29337.534,E2 -29337.534} C_VEL
LIN {X 0,Y 153.212,Z 455.118,A -85,B 0,C 180,E1 -29341.315,E2 -29341.315} C_VEL
LIN {X 0,Y 153.299,Z 456.75,A -85,B 0,C 180,E1 -29343.136,E2 -29343.136} C_VEL
LIN {X 0,Y 148.96,Z 468.623,A -85,B 0,C 180,E1 -29343.807,E2 -29343.807} C_VEL
LIN {X 0,Y 143.653,Z 479.664,A -85,B 0,C 180,E1 -29344.554,E2 -29344.554} C_VEL
LIN {X 0,Y 137.35,Z 490.172,A -85,B 0,C 180,E1 -29345.583,E2 -29345.583} C_VEL
LIN {X 0,Y 130.084,Z 500.021,A -85,B 0,C 180,E1 -29346.893,E2 -29346.893} C_VEL
LIN {X 0,Y 123.814,Z 507.111,A -85,B 0,C 180,E1 -29348.07,E2 -29348.07} C_VEL
LIN {X 0,Y 119.655,Z 511.183,A -85,B 0,C 180,E1 -29348.603,E2 -29348.603} C_VEL
LIN {X 0,Y 111.995,Z 517.454,A -85,B 0,C 180,E1 -29348.763,E2 -29348.763} C_VEL
LIN {X 0,Y 103.895,Z 523.131,A -85,B 0,C 180,E1 -29349.029,E2 -29349.029} C_VEL
LIN {X 0,Y 99.072,Z 526.205,A -85,B 0,C 180,E1 -29349.847,E2 -29349.847} C_VEL
LIN {X 0,Y 90.011,Z 531.395,A -85,B 0,C 180,E1 -29352.567,E2 -29352.567} C_VEL
LIN {X 0,Y 80.522,Z 535.797,A -85,B 0,C 180,E1 -29356.233,E2 -29356.233} C_VEL
LIN {X 0,Y 74.409,Z 538.11,A -85,B 0,C 180,E1 -29359.167,E2 -29359.167} C_VEL
LIN {X 0,Y 68.535,Z 539.968,A -85,B 0,C 180,E1 -29362.635,E2 -29362.635} C_VEL
LIN {X 0,Y 62.945,Z 541.339,A -85,B 0,C 180,E1 -29366.709,E2 -29366.709} C_VEL
LIN {X 0,Y 52.965,Z 542.859,A -85,B 0,C 180,E1 -29377.227,E2 -29377.227} C_VEL
LIN {X 0,Y 46.424,Z 542.845,A -85,B 0,C 180,E1 -29389.198,E2 -29389.198} C_VEL
LIN {X 0,Y 42.891,Z 541.996,A -85,B 0,C 180,E1 -29400.548,E2 -29400.548} C_VEL
LIN {X 0,Y 41.324,Z 540.911,A -85,B 0,C 180,E1 -29410.107,E2 -29410.107} C_VEL
LIN {X 0,Y 40.87,Z 539.368,A -85,B 0,C 180,E1 -29420.091,E2 -29420.091} C_VEL
LIN {X 0,Y 42.292,Z 536.356,A -85,B 0,C 180,E1 -29434.363,E2 -29434.363} C_VEL
LIN {X 0,Y 45.527,Z 532.113,A -85,B 0,C 180,E1 -29447.976,E2 -29447.976} C_VEL
LIN {X 0,Y 51.553,Z 525.792,A -85,B 0,C 180,E1 -29460.738,E2 -29460.738} C_VEL
LIN {X 0,Y 58.185,Z 518.92,A -85,B 0,C 180,E1 -29469.349,E2 -29469.349} C_VEL
LIN {X 0,Y 65.81,Z 510.319,A -85,B 0,C 180,E1 -29476.118,E2 -29476.118} C_VEL
LIN {X 0,Y 72.741,Z 501.482,A -85,B 0,C 180,E1 -29480.611,E2 -29480.611} C_VEL
LIN {X 0,Y 80.097,Z 490.579,A -85,B 0,C 180,E1 -29484.249,E2 -29484.249} C_VEL
LIN {X 0,Y 85.411,Z 481.105,A -85,B 0,C 180,E1 -29486.415,E2 -29486.415} C_VEL
LIN {X 0,Y 90.661,Z 469.264,A -85,B 0,C 180,E1 -29488.501,E2 -29488.501} C_VEL
LIN {X 0,Y 94.967,Z 456.466,A -85,B 0,C 180,E1 -29490.077,E2 -29490.077} C_VEL
LIN {X 0,Y 98.012,Z 443.528,A -85,B 0,C 180,E1 -29491.132,E2 -29491.132} C_VEL
LIN {X 0,Y 100.133,Z 427.923,A -85,B 0,C 180,E1 -29491.816,E2 -29491.816} C_VEL
LIN {X 0,Y 101.293,Z 417.097,A -85,B 0,C 180,E1 -29492.218,E2 -29492.218} C_VEL
LIN {X 0,Y 99.418,Z 411.954,A -85,B 0,C 180,E1 -29496.227,E2 -29496.227} C_VEL
LIN {X 0,Y 98.073,Z 408.623,A -85,B 0,C 180,E1 -29499.771,E2 -29499.771} C_VEL
LIN {X 0,Y 97.315,Z 406.843,A -85,B 0,C 180,E1 -29502.233,E2 -29502.233} C_VEL
LIN {X 0,Y 96.247,Z 403.957,A -85,B 0,C 180,E1 -29507.345,E2 -29507.345} C_VEL
LIN {X 0,Y 95.705,Z 402.713,A -85,B 0,C 180,E1 -29514.19,E2 -29514.19} C_VEL
LIN {X 0,Y 95.919,Z 402.909,A -85,B 0,C 180,E1 -29518.425,E2 -29518.425} C_VEL
LIN {X 0,Y 96.421,Z 403.923,A -85,B 0,C 180,E1 -29522.088,E2 -29522.088} C_VEL
LIN {X 0,Y 97.897,Z 407.965,A -85,B 0,C 180,E1 -29528.254,E2 -29528.254} C_VEL
LIN {X 0,Y 99.576,Z 412.224,A -85,B 0,C 180,E1 -29532.741,E2 -29532.741} C_VEL
LIN {X 0,Y 101.35,Z 417.206,A -85,B 0,C 180,E1 -29536.51,E2 -29536.51} C_VEL
LIN {X 0,Y 98.492,Z 442.045,A -85,B 0,C 180,E1 -29537.505,E2 -29537.505} C_VEL
LIN {X 0,Y 95.603,Z 455.632,A -85,B 0,C 180,E1 -29538.419,E2 -29538.419} C_VEL
LIN {X 0,Y 91.835,Z 467.548,A -85,B 0,C 180,E1 -29539.577,E2 -29539.577} C_VEL
LIN {X 0,Y 86.701,Z 479.556,A -85,B 0,C 180,E1 -29541.232,E2 -29541.232} C_VEL
LIN {X 0,Y 81.311,Z 489.773,A -85,B 0,C 180,E1 -29543.324,E2 -29543.324} C_VEL
LIN {X 0,Y 74.55,Z 500.373,A -85,B 0,C 180,E1 -29546.427,E2 -29546.427} C_VEL
LIN {X 0,Y 67.458,Z 509.931,A -85,B 0,C 180,E1 -29550.748,E2 -29550.748} C_VEL
LIN {X 0,Y 60.814,Z 517.739,A -85,B 0,C 180,E1 -29556.015,E2 -29556.015} C_VEL
LIN {X 0,Y 53.669,Z 525.363,A -85,B 0,C 180,E1 -29563.935,E2 -29563.935} C_VEL
LIN {X 0,Y 47.655,Z 531.466,A -85,B 0,C 180,E1 -29573.857,E2 -29573.857} C_VEL
LIN {X 0,Y 43.526,Z 536.298,A -85,B 0,C 180,E1 -29586.2,E2 -29586.2} C_VEL
LIN {X 0,Y 41.535,Z 539.98,A -85,B 0,C 180,E1 -29600.266,E2 -29600.266} C_VEL
LIN {X 0,Y 41.396,Z 541.868,A -85,B 0,C 180,E1 -29610.007,E2 -29610.007} C_VEL
LIN {X 0,Y 41.54,Z 543.258,A -85,B 0,C 180,E1 -29619.748,E2 -29619.748} C_VEL
LIN {X 0,Y 42.727,Z 544.232,A -85,B 0,C 180,E1 -29629.213,E2 -29629.213} C_VEL
LIN {X 0,Y 47.952,Z 545.038,A -85,B 0,C 180,E1 -29645.899,E2 -29645.899} C_VEL
LIN {X 0,Y 51.843,Z 544.86,A -85,B 0,C 180,E1 -29652.68,E2 -29652.68} C_VEL
LIN {X 0,Y 61.43,Z 543.305,A -85,B 0,C 180,E1 -29663.218,E2 -29663.218} C_VEL
LIN {X 0,Y 66.862,Z 541.954,A -85,B 0,C 180,E1 -29667.241,E2 -29667.241} C_VEL
LIN {X 0,Y 75.82,Z 538.997,A -85,B 0,C 180,E1 -29672.39,E2 -29672.39} C_VEL
LIN {X 0,Y 84.513,Z 535.295,A -85,B 0,C 180,E1 -29676.176,E2 -29676.176} C_VEL
LIN {X 0,Y 93.91,Z 530.37,A -85,B 0,C 180,E1 -29679.312,E2 -29679.312} C_VEL
LIN {X 0,Y 103.589,Z 524.196,A -85,B 0,C 180,E1 -29681.781,E2 -29681.781} C_VEL
LIN {X 0,Y 113.459,Z 516.526,A -85,B 0,C 180,E1 -29683.77,E2 -29683.77} C_VEL
LIN {X 0,Y 121.794,Z 508.693,A -85,B 0,C 180,E1 -29685.143,E2 -29685.143} C_VEL
LIN {X 0,Y 130.973,Z 498.111,A -85,B 0,C 180,E1 -29686.56,E2 -29686.56} C_VEL
LIN {X 0,Y 138.618,Z 487.307,A -85,B 0,C 180,E1 -29687.424,E2 -29687.424} C_VEL
LIN {X 0,Y 145.364,Z 475.137,A -85,B 0,C 180,E1 -29688.14,E2 -29688.14} C_VEL
LIN {X 0,Y 150.524,Z 463.019,A -85,B 0,C 180,E1 -29688.672,E2 -29688.672} C_VEL
LIN {X 0,Y 150.871,Z 461.668,A -85,B 0,C 180,E1 -29689.262,E2 -29689.262} C_VEL
LIN {X 0,Y 150.845,Z 460.079,A -85,B 0,C 180,E1 -29691.966,E2 -29691.966} C_VEL
LIN {X 0,Y 150.809,Z 459.504,A -85,B 0,C 180,E1 -29694.653,E2 -29694.653} C_VEL
LIN {X 0,Y 150.887,Z 459.646,A -85,B 0,C 180,E1 -29697.331,E2 -29697.331} C_VEL
LIN {X 0,Y 150.824,Z 461.573,A -85,B 0,C 180,E1 -29700.668,E2 -29700.668} C_VEL
LIN {X 0,Y 146.747,Z 471.622,A -85,B 0,C 180,E1 -29701.239,E2 -29701.239} C_VEL
LIN {X 0,Y 141.52,Z 481.788,A -85,B 0,C 180,E1 -29701.903,E2 -29701.903} C_VEL
LIN {X 0,Y 134.585,Z 492.594,A -85,B 0,C 180,E1 -29702.885,E2 -29702.885} C_VEL
LIN {X 0,Y 126.829,Z 502.417,A -85,B 0,C 180,E1 -29704.08,E2 -29704.08} C_VEL
LIN {X 0,Y 118.277,Z 511.322,A -85,B 0,C 180,E1 -29705.549,E2 -29705.549} C_VEL
LIN {X 0,Y 109.05,Z 519.23,A -85,B 0,C 180,E1 -29707.407,E2 -29707.407} C_VEL
LIN {X 0,Y 99.072,Z 526.205,A -85,B 0,C 180,E1 -29709.847,E2 -29709.847} C_VEL
LIN {X 0,Y 94.127,Z 529.083,A -85,B 0,C 180,E1 -29710.791,E2 -29710.791} C_VEL
LIN {X 0,Y 85.238,Z 533.32,A -85,B 0,C 180,E1 -29711.568,E2 -29711.568} C_VEL
LIN {X 0,Y 76.123,Z 536.843,A -85,B 0,C 180,E1 -29712.658,E2 -29712.658} C_VEL
LIN {X 0,Y 70.897,Z 538.529,A -85,B 0,C 180,E1 -29714.318,E2 -29714.318} C_VEL
LIN {X 0,Y 66.057,Z 540.003,A -85,B 0,C 180,E1 -29716.743,E2 -29716.743} C_VEL
LIN {X 0,Y 59.621,Z 541.502,A -85,B 0,C 180,E1 -29720.711,E2 -29720.711} C_VEL
LIN {X 0,Y 48.877,Z 543.015,A -85,B 0,C 180,E1 -29730.363,E2 -29730.363} C_VEL
LIN {X 0,Y 40.575,Z 543.023,A -85,B 0,C 180,E1 -29743.859,E2 -29743.859} C_VEL
LIN {X 0,Y 36.728,Z 542.28,A -85,B 0,C 180,E1 -29754.957,E2 -29754.957} C_VEL
LIN {X 0,Y 34.585,Z 541.229,A -85,B 0,C 180,E1 -29766.011,E2 -29766.011} C_VEL
LIN {X 0,Y 33.787,Z 539.748,A -85,B 0,C 180,E1 -29777.986,E2 -29777.986} C_VEL
LIN {X 0,Y 35.393,Z 536.448,A -85,B 0,C 180,E1 -29796.832,E2 -29796.832} C_VEL
LIN {X 0,Y 38.836,Z 532.629,A -85,B 0,C 180,E1 -29811.211,E2 -29811.211} C_VEL
LIN {X 0,Y 45.603,Z 526.387,A -85,B 0,C 180,E1 -29825.296,E2 -29825.296} C_VEL
LIN {X 0,Y 52.895,Z 519.602,A -85,B 0,C 180,E1 -29834.222,E2 -29834.222} C_VEL
LIN {X 0,Y 61.105,Z 511.158,A -85,B 0,C 180,E1 -29840.919,E2 -29840.919} C_VEL
LIN {X 0,Y 68.464,Z 502.447,A -85,B 0,C 180,E1 -29845.198,E2 -29845.198} C_VEL
LIN {X 0,Y 76.159,Z 491.708,A -85,B 0,C 180,E1 -29848.597,E2 -29848.597} C_VEL
LIN {X 0,Y 81.716,Z 482.423,A -85,B 0,C 180,E1 -29850.544,E2 -29850.544} C_VEL
LIN {X 0,Y 87.179,Z 471.002,A -85,B 0,C 180,E1 -29852.461,E2 -29852.461} C_VEL
LIN {X 0,Y 91.817,Z 458.188,A -85,B 0,C 180,E1 -29853.935,E2 -29853.935} C_VEL
LIN {X 0,Y 95.142,Z 445.142,A -85,B 0,C 180,E1 -29854.966,E2 -29854.966} C_VEL
LIN {X 0,Y 97.104,Z 432.787,A -85,B 0,C 180,E1 -29855.514,E2 -29855.514} C_VEL
LIN {X 0,Y 98.449,Z 420.563,A -85,B 0,C 180,E1 -29855.955,E2 -29855.955} C_VEL
LIN {X 0,Y 96.967,Z 415.942,A -85,B 0,C 180,E1 -29860.166,E2 -29860.166} C_VEL
LIN {X 0,Y 95.977,Z 413.355,A -85,B 0,C 180,E1 -29863.778,E2 -29863.778} C_VEL
LIN {X 0,Y 95.197,Z 410.81,A -85,B 0,C 180,E1 -29868.402,E2 -29868.402} C_VEL
LIN {X 0,Y 94.832,Z 409.769,A -85,B 0,C 180,E1 -29874.137,E2 -29874.137} C_VEL
LIN {X 0,Y 94.993,Z 409.894,A -85,B 0,C 180,E1 -29877.879,E2 -29877.879} C_VEL
LIN {X 0,Y 95.379,Z 410.946,A -85,B 0,C 180,E1 -29881.319,E2 -29881.319} C_VEL
LIN {X 0,Y 96.6,Z 414.777,A -85,B 0,C 180,E1 -29887.183,E2 -29887.183} C_VEL
LIN {X 0,Y 98.195,Z 419.667,A -85,B 0,C 180,E1 -29892.005,E2 -29892.005} C_VEL
LIN {X 0,Y 98.517,Z 420.698,A -85,B 0,C 180,E1 -29892.823,E2 -29892.823} C_VEL
LIN {X 0,Y 95.893,Z 442.205,A -85,B 0,C 180,E1 -29893.615,E2 -29893.615} C_VEL
LIN {X 0,Y 92.875,Z 455.794,A -85,B 0,C 180,E1 -29894.444,E2 -29894.444} C_VEL
LIN {X 0,Y 89.192,Z 467.056,A -85,B 0,C 180,E1 -29895.423,E2 -29895.423} C_VEL
LIN {X 0,Y 84.392,Z 478.16,A -85,B 0,C 180,E1 -29896.738,E2 -29896.738} C_VEL
LIN {X 0,Y 77.96,Z 489.894,A -85,B 0,C 180,E1 -29898.829,E2 -29898.829} C_VEL
LIN {X 0,Y 70.882,Z 500.439,A -85,B 0,C 180,E1 -29901.649,E2 -29901.649} C_VEL
LIN {X 0,Y 64.095,Z 509.07,A -85,B 0,C 180,E1 -29905.241,E2 -29905.241} C_VEL
LIN {X 0,Y 56.87,Z 517.003,A -85,B 0,C 180,E1 -29910.122,E2 -29910.122} C_VEL
LIN {X 0,Y 50.194,Z 523.576,A -85,B 0,C 180,E1 -29916.391,E2 -29916.391} C_VEL
LIN {X 0,Y 44.265,Z 529.025,A -85,B 0,C 180,E1 -29924.411,E2 -29924.411} C_VEL
LIN {X 0,Y 38.544,Z 534.344,A -85,B 0,C 180,E1 -29936.847,E2 -29936.847} C_VEL
LIN {X 0,Y 35.11,Z 538.468,A -85,B 0,C 180,E1 -29952.536,E2 -29952.536} C_VEL
LIN {X 0,Y 34.295,Z 541.501,A -85,B 0,C 180,E1 -29970.009,E2 -29970.009} C_VEL
LIN {X 0,Y 34.55,Z 542.95,A -85,B 0,C 180,E1 -29981.745,E2 -29981.745} C_VEL
LIN {X 0,Y 36.073,Z 543.957,A -85,B 0,C 180,E1 -29992.942,E2 -29992.942} C_VEL
LIN {X 0,Y 42.379,Z 544.823,A -85,B 0,C 180,E1 -30011.564,E2 -30011.564} C_VEL
LIN {X 0,Y 46.865,Z 544.693,A -85,B 0,C 180,E1 -30018.583,E2 -30018.583} C_VEL
LIN {X 0,Y 57.45,Z 543.212,A -85,B 0,C 180,E1 -30028.915,E2 -30028.915} C_VEL
LIN {X 0,Y 69.335,Z 540.177,A -85,B 0,C 180,E1 -30035.829,E2 -30035.829} C_VEL
LIN {X 0,Y 78.712,Z 536.752,A -85,B 0,C 180,E1 -30039.648,E2 -30039.648} C_VEL
LIN {X 0,Y 88.364,Z 532.277,A -85,B 0,C 180,E1 -30042.642,E2 -30042.642} C_VEL
LIN {X 0,Y 99.93,Z 525.533,A -85,B 0,C 180,E1 -30045.254,E2 -30045.254} C_VEL
LIN {X 0,Y 110.006,Z 518.212,A -85,B 0,C 180,E1 -30046.987,E2 -30046.987} C_VEL
LIN {X 0,Y 118.466,Z 510.779,A -85,B 0,C 180,E1 -30048.208,E2 -30048.208} C_VEL
LIN {X 0,Y 127.816,Z 500.825,A -85,B 0,C 180,E1 -30049.386,E2 -30049.386} C_VEL
LIN {X 0,Y 135.528,Z 490.665,A -85,B 0,C 180,E1 -30050.164,E2 -30050.164} C_VEL
LIN {X 0,Y 142.421,Z 479.404,A -85,B 0,C 180,E1 -30050.737,E2 -30050.737} C_VEL
LIN {X 0,Y 147.766,Z 468.33,A -85,B 0,C 180,E1 -30051.178,E2 -30051.178} C_VEL
LIN {X 0,Y 148.265,Z 466.938,A -85,B 0,C 180,E1 -30051.825,E2 -30051.825} C_VEL
LIN {X 0,Y 148.312,Z 466.18,A -85,B 0,C 180,E1 -30054.562,E2 -30054.562} C_VEL
LIN {X 0,Y 148.326,Z 466.402,A -85,B 0,C 180,E1 -30057.285,E2 -30057.285} C_VEL
LIN {X 0,Y 147.654,Z 468.23,A -85,B 0,C 180,E1 -30058.329,E2 -30058.329} C_VEL
LIN {X 0,Y 141.889,Z 479.975,A -85,B 0,C 180,E1 -30058.893,E2 -30058.893} C_VEL
LIN {X 0,Y 135.295,Z 490.6,A -85,B 0,C 180,E1 -30059.667,E2 -30059.667} C_VEL
LIN {X 0,Y 127.97,Z 500.185,A -85,B 0,C 180,E1 -30060.626,E2 -30060.626} C_VEL
LIN {X 0,Y 119.536,Z 509.209,A -85,B 0,C 180,E1 -30061.756,E2 -30061.756} C_VEL
LIN {X 0,Y 109.45,Z 518.035,A -85,B 0,C 180,E1 -30063.385,E2 -30063.385} C_VEL
LIN {X 0,Y 98.847,Z 525.541,A -85,B 0,C 180,E1 -30065.476,E2 -30065.476} C_VEL
LIN {X 0,Y 88.709,Z 531.272,A -85,B 0,C 180,E1 -30067.959,E2 -30067.959} C_VEL
LIN {X 0,Y 78.787,Z 535.749,A -85,B 0,C 180,E1 -30071.103,E2 -30071.103} C_VEL
LIN {X 0,Y 70.897,Z 538.529,A -85,B 0,C 180,E1 -30074.318,E2 -30074.318} C_VEL
LIN {X 0,Y 65.652,Z 540.065,A -85,B 0,C 180,E1 -30076.275,E2 -30076.275} C_VEL
LIN {X 0,Y 56.261,Z 541.943,A -85,B 0,C 180,E1 -30078.72,E2 -30078.72} C_VEL
LIN {X 0,Y 46.921,Z 543.091,A -85,B 0,C 180,E1 -30082.188,E2 -30082.188} C_VEL
LIN {X 0,Y 41.959,Z 543.319,A -85,B 0,C 180,E1 -30086.296,E2 -30086.296} C_VEL
LIN {X 0,Y 35.145,Z 543.193,A -85,B 0,C 180,E1 -30096.867,E2 -30096.867} C_VEL
LIN {X 0,Y 31.037,Z 542.566,A -85,B 0,C 180,E1 -30107.196,E2 -30107.196} C_VEL
LIN {X 0,Y 28.104,Z 541.545,A -85,B 0,C 180,E1 -30119.979,E2 -30119.979} C_VEL
LIN {X 0,Y 26.755,Z 540.12,A -85,B 0,C 180,E1 -30134.76,E2 -30134.76} C_VEL
LIN {X 0,Y 28.57,Z 536.581,A -85,B 0,C 180,E1 -30160.252,E2 -30160.252} C_VEL
LIN {X 0,Y 32.318,Z 533.127,A -85,B 0,C 180,E1 -30175.77,E2 -30175.77} C_VEL
LIN {X 0,Y 40.026,Z 526.982,A -85,B 0,C 180,E1 -30191.171,E2 -30191.171} C_VEL
LIN {X 0,Y 48.074,Z 520.284,A -85,B 0,C 180,E1 -30200.121,E2 -30200.121} C_VEL
LIN {X 0,Y 56.903,Z 511.976,A -85,B 0,C 180,E1 -30206.469,E2 -30206.469} C_VEL
LIN {X 0,Y 64.672,Z 503.416,A -85,B 0,C 180,E1 -30210.376,E2 -30210.376} C_VEL
LIN {X 0,Y 72.717,Z 492.831,A -85,B 0,C 180,E1 -30213.37,E2 -30213.37} C_VEL
LIN {X 0,Y 78.477,Z 483.742,A -85,B 0,C 180,E1 -30215.049,E2 -30215.049} C_VEL
LIN {X 0,Y 84.149,Z 472.596,A -85,B 0,C 180,E1 -30216.726,E2 -30216.726} C_VEL
LIN {X 0,Y 89.038,Z 460.137,A -85,B 0,C 180,E1 -30218.031,E2 -30218.031} C_VEL
LIN {X 0,Y 92.733,Z 446.651,A -85,B 0,C 180,E1 -30219.008,E2 -30219.008} C_VEL
LIN {X 0,Y 95.035,Z 433.077,A -85,B 0,C 180,E1 -30219.56,E2 -30219.56} C_VEL
LIN {X 0,Y 96.026,Z 424.256,A -85,B 0,C 180,E1 -30219.881,E2 -30219.881} C_VEL
LIN {X 0,Y 94.959,Z 420.507,A -85,B 0,C 180,E1 -30224.171,E2 -30224.171} C_VEL
LIN {X 0,Y 94.181,Z 417.65,A -85,B 0,C 180,E1 -30229.483,E2 -30229.483} C_VEL
LIN {X 0,Y 94,Z 416.706,A -85,B 0,C 180,E1 -30235.711,E2 -30235.711} C_VEL
LIN {X 0,Y 94.308,Z 417.629,A -85,B 0,C 180,E1 -30239.999,E2 -30239.999} C_VEL
LIN {X 0,Y 95.211,Z 421.198,A -85,B 0,C 180,E1 -30245.559,E2 -30245.559} C_VEL
LIN {X 0,Y 96.077,Z 424.376,A -85,B 0,C 180,E1 -30248.905,E2 -30248.905} C_VEL
LIN {X 0,Y 93.654,Z 442.974,A -85,B 0,C 180,E1 -30249.568,E2 -30249.568} C_VEL
LIN {X 0,Y 90.544,Z 456.243,A -85,B 0,C 180,E1 -30250.275,E2 -30250.275} C_VEL
LIN {X 0,Y 86.635,Z 467.614,A -85,B 0,C 180,E1 -30251.113,E2 -30251.113} C_VEL
LIN {X 0,Y 81.783,Z 478.355,A -85,B 0,C 180,E1 -30252.196,E2 -30252.196} C_VEL
LIN {X 0,Y 75.13,Z 490.016,A -85,B 0,C 180,E1 -30253.963,E2 -30253.963} C_VEL
LIN {X 0,Y 67.757,Z 500.506,A -85,B 0,C 180,E1 -30256.392,E2 -30256.392} C_VEL
LIN {X 0,Y 59.816,Z 509.941,A -85,B 0,C 180,E1 -30259.973,E2 -30259.973} C_VEL
LIN {X 0,Y 52.15,Z 517.676,A -85,B 0,C 180,E1 -30264.557,E2 -30264.557} C_VEL
LIN {X 0,Y 43.567,Z 525.243,A -85,B 0,C 180,E1 -30272.138,E2 -30272.138} C_VEL
LIN {X 0,Y 34.818,Z 532.199,A -85,B 0,C 180,E1 -30285.064,E2 -30285.064} C_VEL
LIN {X 0,Y 29.527,Z 536.778,A -85,B 0,C 180,E1 -30301.584,E2 -30301.584} C_VEL
LIN {X 0,Y 27.623,Z 539.18,A -85,B 0,C 180,E1 -30315.271,E2 -30315.271} C_VEL
LIN {X 0,Y 27.21,Z 541.134,A -85,B 0,C 180,E1 -30330.011,E2 -30330.011} C_VEL
LIN {X 0,Y 27.634,Z 542.628,A -85,B 0,C 180,E1 -30344.744,E2 -30344.744} C_VEL
LIN {X 0,Y 29.648,Z 543.682,A -85,B 0,C 180,E1 -30358.311,E2 -30358.311} C_VEL
LIN {X 0,Y 37.344,Z 544.608,A -85,B 0,C 180,E1 -30378.844,E2 -30378.844} C_VEL
LIN {X 0,Y 48.159,Z 544.025,A -85,B 0,C 180,E1 -30391.127,E2 -30391.127} C_VEL
LIN {X 0,Y 60.356,Z 541.831,A -85,B 0,C 180,E1 -30398.688,E2 -30398.688} C_VEL
LIN {X 0,Y 68.857,Z 539.501,A -85,B 0,C 180,E1 -30402.171,E2 -30402.171} C_VEL
LIN {X 0,Y 79.838,Z 535.437,A -85,B 0,C 180,E1 -30405.55,E2 -30405.55} C_VEL
LIN {X 0,Y 89.885,Z 530.657,A -85,B 0,C 180,E1 -30407.799,E2 -30407.799} C_VEL
LIN {X 0,Y 101.775,Z 523.527,A -85,B 0,C 180,E1 -30409.758,E2 -30409.758} C_VEL
LIN {X 0,Y 112.067,Z 515.767,A -85,B 0,C 180,E1 -30411.025,E2 -30411.025} C_VEL
LIN {X 0,Y 120.667,Z 507.871,A -85,B 0,C 180,E1 -30411.957,E2 -30411.957} C_VEL
LIN {X 0,Y 129.295,Z 498.258,A -85,B 0,C 180,E1 -30412.761,E2 -30412.761} C_VEL
LIN {X 0,Y 137.111,Z 487.577,A -85,B 0,C 180,E1 -30413.289,E2 -30413.289} C_VEL
LIN {X 0,Y 143.648,Z 476.354,A -85,B 0,C 180,E1 -30413.704,E2 -30413.704} C_VEL
LIN {X 0,Y 144.714,Z 474.2,A -85,B 0,C 180,E1 -30413.768,E2 -30413.768} C_VEL
LIN {X 0,Y 145.413,Z 472.711,A -85,B 0,C 180,E1 -30414.454,E2 -30414.454} C_VEL
LIN {X 0,Y 145.396,Z 472.709,A -85,B 0,C 180,E1 -30415.327,E2 -30415.327} C_VEL
LIN {X 0,Y 144.471,Z 474.587,A -85,B 0,C 180,E1 -30415.791,E2 -30415.791} C_VEL
LIN {X 0,Y 138.212,Z 485.712,A -85,B 0,C 180,E1 -30416.325,E2 -30416.325} C_VEL
LIN {X 0,Y 130.728,Z 496.316,A -85,B 0,C 180,E1 -30417.087,E2 -30417.087} C_VEL
LIN {X 0,Y 123.078,Z 505.155,A -85,B 0,C 180,E1 -30417.883,E2 -30417.883} C_VEL
LIN {X 0,Y 114.229,Z 513.601,A -85,B 0,C 180,E1 -30418.913,E2 -30418.913} C_VEL
LIN {X 0,Y 103.669,Z 521.83,A -85,B 0,C 180,E1 -30420.378,E2 -30420.378} C_VEL
LIN {X 0,Y 94.932,Z 527.386,A -85,B 0,C 180,E1 -30421.859,E2 -30421.859} C_VEL
LIN {X 0,Y 84.549,Z 532.784,A -85,B 0,C 180,E1 -30424.032,E2 -30424.032} C_VEL
LIN {X 0,Y 74.323,Z 536.957,A -85,B 0,C 180,E1 -30426.814,E2 -30426.814} C_VEL
LIN {X 0,Y 64.327,Z 540.026,A -85,B 0,C 180,E1 -30430.467,E2 -30430.467} C_VEL
LIN {X 0,Y 56.484,Z 541.761,A -85,B 0,C 180,E1 -30434.411,E2 -30434.411} C_VEL
LIN {X 0,Y 45.61,Z 543.172,A -85,B 0,C 180,E1 -30442.387,E2 -30442.387} C_VEL
LIN {X 0,Y 41.959,Z 543.319,A -85,B 0,C 180,E1 -30446.296,E2 -30446.296} C_VEL
LIN {X 0,Y 37.239,Z 543.386,A -85,B 0,C 180,E1 -30451.453,E2 -30451.453} C_VEL
LIN {X 0,Y 28.918,Z 542.895,A -85,B 0,C 180,E1 -30460.866,E2 -30460.866} C_VEL
LIN {X 0,Y 22.978,Z 541.897,A -85,B 0,C 180,E1 -30472.536,E2 -30472.536} C_VEL
LIN {X 0,Y 20.137,Z 540.738,A -85,B 0,C 180,E1 -30486.134,E2 -30486.134} C_VEL
LIN {X 0,Y 19.731,Z 540.267,A -85,B 0,C 180,E1 -30491.546,E2 -30491.546} C_VEL
LIN {X 0,Y 21.938,Z 536.68,A -85,B 0,C 180,E1 -30526.022,E2 -30526.022} C_VEL
LIN {X 0,Y 28.356,Z 532.044,A -85,B 0,C 180,E1 -30548.274,E2 -30548.274} C_VEL
LIN {X 0,Y 37.856,Z 525.555,A -85,B 0,C 180,E1 -30562.081,E2 -30562.081} C_VEL
LIN {X 0,Y 46.958,Z 518.442,A -85,B 0,C 180,E1 -30569.368,E2 -30569.368} C_VEL
LIN {X 0,Y 56.544,Z 509.578,A -85,B 0,C 180,E1 -30574.292,E2 -30574.292} C_VEL
LIN {X 0,Y 64.795,Z 500.47,A -85,B 0,C 180,E1 -30577.201,E2 -30577.201} C_VEL
LIN {X 0,Y 72.356,Z 490.368,A -85,B 0,C 180,E1 -30579.196,E2 -30579.196} C_VEL
LIN {X 0,Y 78.285,Z 480.715,A -85,B 0,C 180,E1 -30580.486,E2 -30580.486} C_VEL
LIN {X 0,Y 84.128,Z 468.594,A -85,B 0,C 180,E1 -30581.84,E2 -30581.84} C_VEL
LIN {X 0,Y 88.618,Z 456.277,A -85,B 0,C 180,E1 -30582.779,E2 -30582.779} C_VEL
LIN {X 0,Y 91.707,Z 444.181,A -85,B 0,C 180,E1 -30583.426,E2 -30583.426} C_VEL
LIN {X 0,Y 94.036,Z 428.397,A -85,B 0,C 180,E1 -30583.931,E2 -30583.931} C_VEL
LIN {X 0,Y 93.49,Z 426.232,A -85,B 0,C 180,E1 -30587.226,E2 -30587.226} C_VEL
LIN {X 0,Y 93.184,Z 424.481,A -85,B 0,C 180,E1 -30590.752,E2 -30590.752} C_VEL
LIN {X 0,Y 93.124,Z 423.76,A -85,B 0,C 180,E1 -30595.671,E2 -30595.671} C_VEL
LIN {X 0,Y 93.31,Z 424.592,A -85,B 0,C 180,E1 -30599.108,E2 -30599.108} C_VEL
LIN {X 0,Y 94.003,Z 428.006,A -85,B 0,C 180,E1 -30604.421,E2 -30604.421} C_VEL
LIN {X 0,Y 94.084,Z 428.466,A -85,B 0,C 180,E1 -30604.89,E2 -30604.89} C_VEL
LIN {X 0,Y 91.758,Z 444.498,A -85,B 0,C 180,E1 -30605.354,E2 -30605.354} C_VEL
LIN {X 0,Y 88.368,Z 457.701,A -85,B 0,C 180,E1 -30605.94,E2 -30605.94} C_VEL
LIN {X 0,Y 84.014,Z 469.45,A -85,B 0,C 180,E1 -30606.634,E2 -30606.634} C_VEL
